C01812=1021.394,-73.795,405.018,166.174,50.269,159.076
C01813=1021.400,-73.545,405.007,166.177,50.265,159.076
C01814=1021.405,-73.295,404.997,166.180,50.261,159.076
C01815=1021.410,-73.046,404.986,166.182,50.257,159.076
C01816=1021.416,-72.796,404.976,166.185,50.253,159.075
C01817=1021.423,-72.475,404.962,166.189,50.248,159.075
C01818=1021.430,-72.155,404.949,166.193,50.243,159.075
C01819=1021.437,-71.835,404.935,166.198,50.238,159.075
C01820=1021.444,-71.515,404.921,166.201,50.233,159.074
C01821=1021.449,-71.265,404.910,166.204,50.228,159.074
C01822=1021.454,-71.015,404.900,166.207,50.225,159.074
C01823=1021.460,-70.766,404.889,166.210,50.221,159.074
C01824=1021.466,-70.516,404.878,166.213,50.217,159.073
C01825=1021.471,-70.286,404.869,166.216,50.213,159.073
C01826=1021.476,-70.056,404.859,166.219,50.209,159.073
C01827=1021.481,-69.826,404.849,166.221,50.206,159.073
C01828=1021.487,-69.597,404.839,166.224,50.202,159.073
C01829=1021.492,-69.367,404.829,166.227,50.199,159.072
C01830=1021.497,-69.138,404.820,166.229,50.195,159.072
C01831=1021.502,-68.907,404.809,166.232,50.191,159.072
C01832=1021.507,-68.677,404.800,166.235,50.187,159.072
C01833=1021.513,-68.428,404.789,166.238,50.184,159.072
C01834=1021.518,-68.178,404.778,166.241,50.180,159.071
C01835=1021.524,-67.928,404.768,166.243,50.176,159.071
C01836=1021.530,-67.679,404.757,166.247,50.171,159.071
C01837=1021.535,-67.429,404.746,166.250,50.167,159.071
C01838=1021.541,-67.180,404.735,166.253,50.164,159.071
C01839=1021.546,-66.930,404.725,166.256,50.160,159.070
C01840=1021.552,-66.680,404.714,166.259,50.155,159.070
C01841=1021.558,-66.431,404.703,166.262,50.151,159.070
C01842=1021.564,-66.181,404.692,166.265,50.147,159.070
C01843=1021.569,-65.932,404.681,166.268,50.144,159.070
C01844=1021.575,-65.681,404.670,166.272,50.139,159.069
C01845=1021.580,-65.431,404.659,166.274,50.135,159.069
C01846=1021.586,-65.182,404.648,166.277,50.131,159.069
C01847=1021.592,-64.932,404.638,166.280,50.127,159.069
C01848=1021.598,-64.683,404.627,166.282,50.123,159.068
C01849=1021.603,-64.433,404.617,166.286,50.119,159.068
C01850=1021.609,-64.183,404.606,166.289,50.115,159.068
C01851=1021.615,-63.934,404.595,166.292,50.111,159.068
C01852=1021.620,-63.684,404.584,166.294,50.107,159.067
C01853=1021.626,-63.434,404.572,166.298,50.103,159.067
C01854=1021.632,-63.184,404.561,166.301,50.099,159.067
C01855=1021.637,-62.935,404.550,166.304,50.095,159.067
C01856=1021.643,-62.685,404.539,166.306,50.090,159.066
C01857=1021.649,-62.436,404.529,166.310,50.086,159.066
C01858=1021.654,-62.186,404.518,166.313,50.083,159.066
C01859=1021.660,-61.936,404.508,166.316,50.079,159.066
C01860=1021.666,-61.686,404.496,166.318,50.075,159.066
C01861=1021.672,-61.436,404.485,166.322,50.070,159.065
C01862=1021.677,-61.187,404.474,166.325,50.066,159.065
C01863=1021.683,-60.937,404.463,166.328,50.062,159.065
C01864=1021.689,-60.688,404.452,166.330,50.058,159.064
C01865=1021.695,-60.437,404.441,166.334,50.054,159.064
C01866=1021.701,-60.188,404.430,166.337,50.050,159.064
C01867=1021.706,-59.938,404.419,166.339,50.045,159.064
C01868=1021.712,-59.689,404.408,166.343,50.041,159.064
C01869=1021.718,-59.439,404.397,166.346,50.037,159.063
C01870=1021.724,-59.189,404.386,166.349,50.033,159.063
C01871=1021.729,-58.939,404.375,166.352,50.030,159.063
C01872=1021.735,-58.690,404.364,166.355,50.025,159.063
C01873=1021.741,-58.441,404.353,166.358,50.021,159.062
C01874=1021.747,-58.190,404.342,166.361,50.017,159.062
C01875=1021.753,-57.941,404.331,166.363,50.013,159.062
C01876=1021.759,-57.691,404.320,166.367,50.009,159.062
C01877=1021.764,-57.442,404.309,166.370,50.005,159.061
C01878=1021.770,-57.191,404.297,166.373,50.000,159.061
C01879=1021.776,-56.942,404.286,166.375,49.996,159.061
C01880=1021.782,-56.693,404.275,166.379,49.992,159.061
C01881=1021.788,-56.443,404.264,166.382,49.988,159.060
C01882=1021.794,-56.193,404.253,166.384,49.984,159.060
C01883=1021.799,-55.944,404.242,166.388,49.980,159.060
C01884=1021.804,-55.694,404.230,166.391,49.975,159.060
C01885=1021.811,-55.444,404.219,166.394,49.971,159.059
C01886=1021.817,-55.194,404.208,166.396,49.967,159.059
C01887=1021.822,-54.945,404.197,166.400,49.963,159.059
C01888=1021.829,-54.695,404.185,166.403,49.959,159.059
C01889=1021.835,-54.446,404.174,166.405,49.955,159.058
C01890=1021.840,-54.196,404.164,166.409,49.950,159.058
C01891=1021.846,-53.946,404.152,166.412,49.946,159.058
C01892=1021.852,-53.696,404.141,166.414,49.942,159.057
C01893=1021.859,-53.417,404.128,166.418,49.937,159.057
C01894=1021.866,-53.138,404.116,166.421,49.932,159.057
C01895=1021.872,-52.859,404.103,166.424,49.928,159.057
C01896=1021.879,-52.579,404.091,166.427,49.923,159.056
C01897=1021.885,-52.330,404.079,166.431,49.919,159.056
C01898=1021.890,-52.080,404.068,166.434,49.915,159.056
C01899=1021.897,-51.830,404.057,166.437,49.911,159.055
C01900=1021.902,-51.580,404.045,166.439,49.907,159.055
C01901=1021.908,-51.331,404.033,166.443,49.902,159.055
C01902=1021.914,-51.081,404.023,166.446,49.898,159.055
C01903=1021.920,-50.832,404.012,166.448,49.894,159.054
C01904=1021.926,-50.582,403.999,166.451,49.890,159.054
C01905=1021.932,-50.332,403.988,166.455,49.886,159.054
C01906=1021.937,-50.082,403.976,166.458,49.882,159.054
C01907=1021.943,-49.833,403.965,166.460,49.878,159.053
C01908=1021.949,-49.583,403.953,166.463,49.874,159.053
C01909=1021.955,-49.334,403.941,166.466,49.870,159.053
C01910=1021.960,-49.084,403.930,166.469,49.866,159.053
C01911=1021.966,-48.834,403.917,166.473,49.862,159.052
C01912=1021.971,-48.584,403.906,166.475,49.858,159.052
C01913=1021.977,-48.335,403.894,166.478,49.854,159.052
C01914=1021.983,-48.085,403.883,166.481,49.850,159.052
C01915=1021.989,-47.835,403.870,166.484,49.846,159.051
C01916=1021.995,-47.586,403.860,166.486,49.842,159.051
C01917=1022.000,-47.337,403.847,166.490,49.838,159.051
C01918=1022.006,-47.086,403.836,166.493,49.834,159.051
C01919=1022.012,-46.837,403.824,166.496,49.830,159.050
C01920=1022.017,-46.587,403.812,166.498,49.826,159.050
C01921=1022.023,-46.338,403.801,166.501,49.822,159.050
C01922=1022.029,-46.088,403.788,166.504,49.818,159.050
C01923=1022.035,-45.838,403.777,166.508,49.814,159.050
C01924=1022.041,-45.589,403.765,166.511,49.810,159.049
C01925=1022.047,-45.339,403.754,166.513,49.806,159.049
C01926=1022.053,-45.089,403.741,166.516,49.802,159.049
C01927=1022.059,-44.840,403.730,166.519,49.798,159.048
C01928=1022.064,-44.590,403.718,166.521,49.794,159.048
C01929=1022.070,-44.341,403.705,166.525,49.789,159.048
C01930=1022.076,-44.090,403.694,166.528,49.785,159.048
C01931=1022.081,-43.841,403.682,166.531,49.781,159.047
C01932=1022.088,-43.592,403.670,166.533,49.777,159.047
C01933=1022.093,-43.341,403.658,166.536,49.773,159.047
C01934=1022.099,-43.092,403.647,166.540,49.770,159.047
C01935=1022.105,-42.842,403.634,166.543,49.766,159.046
C01936=1022.110,-42.593,403.623,166.546,49.762,159.046
C01937=1022.117,-42.343,403.611,166.548,49.758,159.046
C01938=1022.122,-42.094,403.599,166.551,49.753,159.045
C01939=1022.129,-41.844,403.587,166.554,49.749,159.045
C01940=1022.134,-41.594,403.575,166.558,49.745,159.045
C01941=1022.140,-41.345,403.563,166.560,49.741,159.045
C01942=1022.147,-41.095,403.551,166.563,49.737,159.044
C01943=1022.152,-40.845,403.539,166.566,49.733,159.044
C01944=1022.158,-40.596,403.527,166.568,49.729,159.044
C01945=1022.163,-40.346,403.515,166.572,49.725,159.044
C01946=1022.170,-40.097,403.503,166.575,49.721,159.043
C01947=1022.176,-39.846,403.491,166.578,49.717,159.043
C01948=1022.181,-39.597,403.479,166.580,49.713,159.043
C01949=1022.188,-39.348,403.467,166.583,49.708,159.042
C01950=1022.194,-39.098,403.454,166.587,49.704,159.042
C01951=1022.199,-38.849,403.442,166.589,49.700,159.042
C01952=1022.204,-38.598,403.430,166.592,49.696,159.042
C01953=1022.210,-38.348,403.418,166.595,49.692,159.041
C01954=1022.216,-38.099,403.406,166.598,49.688,159.041
C01955=1022.222,-37.849,403.394,166.601,49.685,159.041
C01956=1022.228,-37.600,403.381,166.603,49.681,159.041
C01957=1022.234,-37.321,403.367,166.607,49.676,159.040
C01958=1022.241,-37.043,403.354,166.610,49.672,159.040
C01959=1022.248,-36.763,403.341,166.613,49.667,159.040
C01960=1022.253,-36.484,403.327,166.617,49.662,159.039
C01961=1022.259,-36.234,403.314,166.620,49.659,159.039
C01962=1022.265,-35.984,403.301,166.623,49.655,159.039
C01963=1022.271,-35.735,403.289,166.625,49.651,159.039
C01964=1022.277,-35.486,403.277,166.628,49.647,159.038
C01965=1022.283,-35.236,403.265,166.631,49.643,159.038
C01966=1022.288,-34.987,403.253,166.633,49.639,159.038
C01967=1022.294,-34.737,403.240,166.636,49.635,159.037
C01968=1022.300,-34.487,403.227,166.640,49.630,159.037
C01969=1022.306,-34.237,403.215,166.643,49.626,159.037
C01970=1022.312,-33.988,403.203,166.645,49.622,159.037
C01971=1022.318,-33.738,403.191,166.648,49.618,159.036
C01972=1022.324,-33.488,403.178,166.651,49.615,159.036
C01973=1022.330,-33.238,403.166,166.654,49.611,159.036
C01974=1022.336,-32.990,403.153,166.657,49.607,159.036
C01975=1022.341,-32.740,403.140,166.659,49.603,159.035
C01976=1022.347,-32.490,403.128,166.663,49.599,159.035
C01977=1022.353,-32.240,403.115,166.666,49.595,159.035
C01978=1022.359,-31.991,403.103,166.669,49.591,159.035
C01979=1022.365,-31.742,403.091,166.671,49.587,159.034
C01980=1022.371,-31.492,403.078,166.674,49.583,159.034
C01981=1022.377,-31.242,403.066,166.677,49.579,159.034
C01982=1022.382,-30.993,403.054,166.679,49.575,159.033
C01983=1022.388,-30.743,403.041,166.682,49.570,159.033
C01984=1022.395,-30.493,403.028,166.686,49.566,159.033
C01985=1022.400,-30.244,403.015,166.689,49.562,159.033
C01986=1022.406,-29.994,403.003,166.691,49.558,159.032
C01987=1022.412,-29.745,402.991,166.694,49.554,159.032
C01988=1022.418,-29.495,402.979,166.697,49.550,159.032
C01989=1022.424,-29.245,402.966,166.700,49.546,159.031
C01990=1022.430,-28.996,402.953,166.702,49.542,159.031
C01991=1022.436,-28.746,402.940,166.706,49.538,159.031
C01992=1022.442,-28.496,402.928,166.709,49.534,159.031
C01993=1022.448,-28.247,402.915,166.711,49.530,159.030
C01994=1022.453,-27.997,402.903,166.714,49.526,159.030
C01995=1022.460,-27.748,402.890,166.717,49.522,159.030
C01996=1022.466,-27.498,402.878,166.720,49.518,159.029
C01997=1022.471,-27.248,402.864,166.722,49.514,159.029
C01998=1022.477,-26.998,402.852,166.725,49.510,159.029
C01999=1022.484,-26.749,402.839,166.728,49.506,159.028
C02000=1022.489,-26.499,402.826,166.731,49.502,159.028
C02001=1022.495,-26.250,402.814,166.734,49.497,159.028
C02002=1022.501,-26.000,402.801,166.737,49.493,159.028
C02003=1022.506,-25.750,402.787,166.740,49.490,159.028
C02004=1022.512,-25.501,402.774,166.743,49.486,159.027
C02005=1022.518,-25.251,402.762,166.746,49.482,159.027
C02006=1022.524,-25.001,402.749,166.748,49.478,159.027
C02007=1022.530,-24.752,402.736,166.751,49.474,159.026
C02008=1022.536,-24.502,402.723,166.754,49.470,159.026
C02009=1022.541,-24.253,402.710,166.757,49.466,159.026
C02010=1022.547,-24.003,402.697,166.759,49.462,159.025
C02011=1022.553,-23.754,402.684,166.762,49.458,159.025
C02012=1022.559,-23.504,402.671,166.765,49.454,159.025
C02013=1022.565,-23.255,402.658,166.768,49.450,159.024
C02014=1022.571,-23.005,402.646,166.770,49.446,159.024
C02015=1022.577,-22.755,402.632,166.773,49.443,159.024
C02016=1022.583,-22.506,402.619,166.776,49.439,159.024
C02017=1022.589,-22.256,402.607,166.779,49.435,159.023
C02018=1022.595,-22.006,402.593,166.783,49.430,159.023
C02019=1022.601,-21.756,402.581,166.785,49.426,159.023
C02020=1022.606,-21.507,402.567,166.788,49.422,159.023
C02021=1022.613,-21.228,402.553,166.790,49.418,159.022
C02022=1022.620,-20.947,402.538,166.794,49.413,159.022
C02023=1022.626,-20.668,402.523,166.797,49.409,159.021
C02024=1022.633,-20.388,402.509,166.800,49.404,159.021
C02025=1022.639,-20.138,402.496,166.803,49.400,159.021
C02026=1022.645,-19.889,402.483,166.806,49.396,159.021
C02027=1022.651,-19.639,402.470,166.809,49.392,159.020
C02028=1022.657,-19.389,402.456,166.811,49.388,159.020
C02029=1022.663,-19.140,402.444,166.814,49.384,159.020
C02030=1022.669,-18.890,402.430,166.817,49.380,159.019
C02031=1022.675,-18.641,402.417,166.820,49.376,159.019
C02032=1022.680,-18.391,402.404,166.823,49.372,159.019
C02033=1022.687,-18.142,402.391,166.826,49.368,159.019
C02034=1022.693,-17.892,402.378,166.829,49.364,159.018
C02035=1022.699,-17.642,402.365,166.832,49.360,159.018
C02036=1022.705,-17.393,402.352,166.834,49.356,159.018
C02037=1022.711,-17.143,402.339,166.837,49.352,159.017
C02038=1022.716,-16.894,402.325,166.840,49.348,159.017
C02039=1022.722,-16.644,402.312,166.842,49.343,159.017
C02040=1022.728,-16.395,402.299,166.845,49.339,159.016
C02041=1022.735,-16.145,402.286,166.848,49.335,159.016
C02042=1022.741,-15.896,402.273,166.850,49.331,159.016
C02043=1022.746,-15.646,402.260,166.853,49.327,159.015
C02044=1022.752,-15.397,402.247,166.856,49.323,159.015
C02045=1022.758,-15.147,402.233,166.859,49.319,159.015
C02046=1022.764,-14.898,402.219,166.862,49.316,159.015
C02047=1022.769,-14.648,402.206,166.864,49.312,159.014
C02048=1022.776,-14.398,402.193,166.867,49.308,159.014
C02049=1022.781,-14.148,402.179,166.870,49.304,159.014
C02050=1022.788,-13.899,402.165,166.873,49.300,159.013
C02051=1022.793,-13.649,402.152,166.875,49.296,159.013
C02052=1022.799,-13.400,402.138,166.878,49.292,159.013
C02053=1022.805,-13.151,402.125,166.881,49.288,159.012
C02054=1022.811,-12.900,402.112,166.884,49.284,159.012
C02055=1022.817,-12.651,402.099,166.886,49.280,159.012
C02056=1022.822,-12.402,402.085,166.889,49.276,159.011
C02057=1022.829,-12.152,402.072,166.892,49.272,159.011
C02058=1022.835,-11.902,402.057,166.895,49.268,159.011
C02059=1022.841,-11.653,402.044,166.897,49.264,159.010
C02060=1022.846,-11.403,402.030,166.900,49.260,159.010
C02061=1022.853,-11.154,402.017,166.903,49.256,159.010
C02062=1022.858,-10.904,402.003,166.906,49.252,159.010
C02063=1022.864,-10.655,401.990,166.908,49.248,159.009
C02064=1022.869,-10.405,401.977,166.911,49.244,159.009
C02065=1022.876,-10.155,401.963,166.915,49.240,159.009
C02066=1022.882,-9.905,401.949,166.918,49.236,159.008
C02067=1022.888,-9.656,401.936,166.920,49.232,159.008
C02068=1022.893,-9.406,401.922,166.923,49.228,159.008
C02069=1022.900,-9.157,401.909,166.926,49.224,159.007
C02070=1022.905,-8.908,401.895,166.929,49.220,159.007
C02071=1022.912,-8.658,401.881,166.931,49.216,159.007
C02072=1022.918,-8.408,401.868,166.934,49.212,159.007
C02073=1022.924,-8.159,401.854,166.937,49.208,159.006
C02074=1022.930,-7.910,401.841,166.940,49.204,159.006
C02075=1022.935,-7.660,401.827,166.942,49.200,159.006
C02076=1022.942,-7.410,401.813,166.945,49.196,159.005
C02077=1022.948,-7.160,401.799,166.948,49.192,159.005
C02078=1022.954,-6.911,401.786,166.951,49.188,159.005
C02079=1022.959,-6.662,401.772,166.953,49.184,159.004
C02080=1022.966,-6.412,401.759,166.956,49.180,159.004
C02081=1022.972,-6.162,401.745,166.959,49.176,159.004
C02082=1022.978,-5.913,401.732,166.962,49.172,159.003
C02083=1022.983,-5.663,401.718,166.964,49.169,159.003
C02084=1022.990,-5.414,401.703,166.967,49.165,159.003
C02085=1022.997,-5.132,401.688,166.970,49.160,159.002
C02086=1023.003,-4.851,401.672,166.973,49.155,159.002
C02087=1023.010,-4.569,401.657,166.977,49.151,159.002
C02088=1023.017,-4.288,401.641,166.979,49.146,159.001
C02089=1023.023,-4.039,401.628,166.982,49.142,159.001
C02090=1023.029,-3.788,401.614,166.985,49.138,159.001
C02091=1023.034,-3.539,401.600,166.987,49.134,159.000
C02092=1023.040,-3.289,401.586,166.990,49.130,159.000
C02093=1023.046,-3.040,401.571,166.993,49.127,159.000
C02094=1023.052,-2.790,401.557,166.996,49.123,158.999
C02095=1023.058,-2.541,401.544,166.999,49.119,158.999
C02096=1023.064,-2.292,401.529,167.002,49.115,158.999
C02097=1023.070,-2.041,401.515,167.003,49.111,158.998
C02098=1023.075,-1.792,401.501,167.006,49.107,158.998
C02099=1023.081,-1.543,401.487,167.009,49.103,158.998
C02100=1023.087,-1.293,401.472,167.012,49.099,158.997
C02101=1023.093,-1.043,401.459,167.014,49.095,158.997
C02102=1023.099,-0.794,401.445,167.017,49.091,158.997
C02103=1023.105,-0.545,401.431,167.020,49.087,158.997
C02104=1023.111,-0.295,401.416,167.023,49.083,158.996
C02105=1023.117,-0.046,401.402,167.026,49.080,158.996
C02106=1023.122,0.204,401.388,167.028,49.076,158.996
C02107=1023.128,0.454,401.374,167.031,49.072,158.995
C02108=1023.134,0.703,401.359,167.034,49.068,158.995
C02109=1023.140,0.952,401.346,167.037,49.064,158.995
C02110=1023.146,1.203,401.332,167.039,49.060,158.994
C02111=1023.152,1.452,401.317,167.041,49.057,158.994
C02112=1023.157,1.701,401.303,167.044,49.053,158.994
C02113=1023.164,1.951,401.288,167.047,49.049,158.993
C02114=1023.169,2.200,401.274,167.049,49.045,158.993
C02115=1023.176,2.450,401.259,167.052,49.041,158.993
C02116=1023.182,2.699,401.246,167.055,49.037,158.992
C02117=1023.187,2.949,401.232,167.058,49.033,158.992
C02118=1023.194,3.199,401.217,167.060,49.029,158.992
C02119=1023.199,3.448,401.204,167.063,49.025,158.991
C02120=1023.205,3.697,401.189,167.066,49.021,158.991
C02121=1023.211,3.947,401.175,167.069,49.017,158.991
C02122=1023.217,4.196,401.160,167.072,49.013,158.991
C02123=1023.223,4.447,401.146,167.074,49.009,158.990
C02124=1023.229,4.695,401.132,167.077,49.005,158.990
C02125=1023.236,4.946,401.118,167.080,49.001,158.990
C02126=1023.241,5.195,401.103,167.083,48.997,158.989
C02127=1023.247,5.444,401.089,167.084,48.994,158.989
C02128=1023.253,5.694,401.074,167.087,48.990,158.989
C02129=1023.259,5.943,401.060,167.089,48.985,158.988
C02130=1023.265,6.193,401.046,167.092,48.981,158.988
C02131=1023.271,6.443,401.032,167.095,48.977,158.987
C02132=1023.278,6.692,401.017,167.098,48.973,158.987
C02133=1023.283,6.941,401.003,167.101,48.969,158.987
C02134=1023.289,7.190,400.989,167.103,48.965,158.986
C02135=1023.295,7.440,400.974,167.106,48.961,158.986
C02136=1023.301,7.690,400.960,167.109,48.957,158.986
C02137=1023.307,7.939,400.945,167.112,48.953,158.985
C02138=1023.313,8.189,400.931,167.114,48.950,158.985
C02139=1023.319,8.439,400.916,167.117,48.946,158.985
C02140=1023.325,8.688,400.902,167.120,48.941,158.984
C02141=1023.332,8.937,400.888,167.122,48.937,158.984
C02142=1023.337,9.186,400.873,167.125,48.933,158.984
C02143=1023.343,9.437,400.859,167.128,48.929,158.983
C02144=1023.349,9.686,400.845,167.131,48.925,158.983
C02145=1023.356,9.935,400.830,167.133,48.921,158.983
C02146=1023.361,10.185,400.816,167.136,48.917,158.982
C02147=1023.367,10.435,400.801,167.139,48.913,158.982
C02148=1023.373,10.684,400.786,167.141,48.909,158.982
C02149=1023.380,10.967,400.770,167.144,48.905,158.981
C02150=1023.387,11.250,400.754,167.148,48.900,158.981
C02151=1023.394,11.534,400.737,167.150,48.895,158.980
C02152=1023.402,11.817,400.721,167.153,48.890,158.980
C02153=1023.407,12.066,400.706,167.156,48.886,158.980
C02154=1023.413,12.317,400.692,167.159,48.882,158.979
C02155=1023.420,12.566,400.677,167.162,48.878,158.979
C02156=1023.426,12.815,400.663,167.164,48.875,158.979
C02157=1023.432,13.066,400.648,167.166,48.871,158.978
C02158=1023.437,13.314,400.634,167.169,48.866,158.978
C02159=1023.444,13.564,400.619,167.172,48.862,158.977
C02160=1023.450,13.814,400.604,167.174,48.858,158.977
C02161=1023.456,14.063,400.589,167.177,48.854,158.977
C02162=1023.462,14.313,400.575,167.180,48.850,158.976
C02163=1023.467,14.562,400.560,167.183,48.846,158.976
C02164=1023.473,14.812,400.545,167.185,48.843,158.976
C02165=1023.479,15.061,400.530,167.188,48.839,158.975
C02166=1023.486,15.311,400.515,167.191,48.835,158.975
C02167=1023.492,15.560,400.500,167.194,48.831,158.975
C02168=1023.498,15.809,400.486,167.195,48.827,158.974
C02169=1023.503,16.059,400.470,167.198,48.823,158.974
C02170=1023.509,16.308,400.456,167.201,48.819,158.974
C02171=1023.515,16.558,400.442,167.204,48.815,158.973
C02172=1023.522,16.808,400.427,167.207,48.811,158.973
C02173=1023.527,17.057,400.412,167.209,48.807,158.973
C02174=1023.533,17.307,400.396,167.212,48.803,158.972
C02175=1023.539,17.556,400.382,167.215,48.799,158.972
C02176=1023.545,17.806,400.367,167.217,48.795,158.972
C02177=1023.552,18.055,400.352,167.220,48.791,158.971
C02178=1023.557,18.304,400.337,167.222,48.787,158.971
C02179=1023.563,18.554,400.322,167.225,48.783,158.971
C02180=1023.569,18.804,400.307,167.227,48.779,158.970
C02181=1023.575,19.053,400.292,167.230,48.776,158.970
C02182=1023.582,19.302,400.277,167.233,48.772,158.970
C02183=1023.588,19.552,400.262,167.236,48.768,158.969
C02184=1023.593,19.801,400.247,167.238,48.763,158.969
C02185=1023.599,20.051,400.232,167.241,48.759,158.968
C02186=1023.606,20.301,400.217,167.243,48.755,158.968
C02187=1023.611,20.550,400.202,167.245,48.752,158.968
C02188=1023.617,20.800,400.187,167.248,48.748,158.967
C02189=1023.624,21.049,400.172,167.251,48.744,158.967
C02190=1023.629,21.298,400.156,167.254,48.740,158.967
C02191=1023.635,21.548,400.142,167.257,48.736,158.966
C02192=1023.642,21.797,400.127,167.259,48.732,158.966
C02193=1023.647,22.046,400.111,167.262,48.728,158.966
C02194=1023.653,22.296,400.096,167.264,48.724,158.965
C02195=1023.659,22.546,400.081,167.267,48.720,158.965
C02196=1023.665,22.795,400.066,167.269,48.716,158.965
C02197=1023.671,23.044,400.051,167.272,48.713,158.964
C02198=1023.677,23.294,400.035,167.275,48.708,158.964
C02199=1023.683,23.544,400.020,167.277,48.704,158.963
C02200=1023.689,23.793,400.006,167.280,48.700,158.963
C02201=1023.695,24.043,399.990,167.283,48.696,158.963
C02202=1023.701,24.292,399.975,167.285,48.693,158.962
C02203=1023.707,24.541,399.960,167.288,48.689,158.962
C02204=1023.713,24.791,399.944,167.290,48.685,158.962
C02205=1023.719,25.040,399.929,167.293,48.681,158.961
C02206=1023.726,25.290,399.914,167.296,48.676,158.961
C02207=1023.731,25.539,399.899,167.298,48.672,158.961
C02208=1023.737,25.788,399.884,167.301,48.668,158.960
C02209=1023.743,26.038,399.868,167.304,48.664,158.960
C02210=1023.749,26.288,399.853,167.307,48.661,158.960
C02211=1023.755,26.537,399.838,167.308,48.657,158.959
C02212=1023.761,26.786,399.822,167.311,48.653,158.959
C02213=1023.768,27.071,399.805,167.315,48.648,158.958
C02214=1023.775,27.356,399.788,167.317,48.643,158.958
C02215=1023.782,27.641,399.770,167.321,48.639,158.958
C02216=1023.788,27.926,399.753,167.323,48.635,158.957
C02217=1023.795,28.175,399.737,167.326,48.631,158.957
C02218=1023.801,28.425,399.722,167.329,48.627,158.956
C02219=1023.806,28.675,399.706,167.331,48.623,158.956
C02220=1023.813,28.923,399.691,167.334,48.619,158.956
C02221=1023.818,29.173,399.675,167.336,48.615,158.955
C02222=1023.825,29.422,399.659,167.339,48.611,158.955
C02223=1023.831,29.672,399.644,167.342,48.608,158.955
C02224=1023.836,29.922,399.628,167.344,48.603,158.954
C02225=1023.842,30.170,399.613,167.346,48.599,158.954
C02226=1023.848,30.420,399.598,167.349,48.595,158.953
C02227=1023.855,30.669,399.582,167.352,48.591,158.953
C02228=1023.860,30.919,399.566,167.355,48.588,158.953
C02229=1023.866,31.169,399.550,167.357,48.584,158.952
C02230=1023.873,31.418,399.535,167.360,48.580,158.952
C02231=1023.878,31.667,399.519,167.362,48.576,158.952
C02232=1023.884,31.917,399.504,167.365,48.572,158.951
C02233=1023.890,32.166,399.488,167.367,48.568,158.951
C02234=1023.896,32.416,399.473,167.370,48.564,158.951
C02235=1023.903,32.665,399.457,167.373,48.560,158.950
C02236=1023.908,32.915,399.441,167.375,48.556,158.950
C02237=1023.914,33.163,399.426,167.378,48.552,158.950
C02238=1023.920,33.413,399.410,167.380,48.548,158.949
C02239=1023.926,33.663,399.394,167.383,48.544,158.949
C02240=1023.932,33.912,399.379,167.386,48.541,158.948
C02241=1023.938,34.162,399.363,167.388,48.537,158.948
C02242=1023.944,34.412,399.347,167.391,48.532,158.948
C02243=1023.951,34.661,399.332,167.394,48.528,158.947
C02244=1023.956,34.911,399.316,167.395,48.525,158.947
C02245=1023.963,35.160,399.301,167.398,48.521,158.946
C02246=1023.968,35.409,399.285,167.401,48.517,158.946
C02247=1023.974,35.658,399.269,167.404,48.513,158.946
C02248=1023.981,35.907,399.254,167.406,48.508,158.945
C02249=1023.986,36.157,399.238,167.409,48.504,158.945
C02250=1023.993,36.406,399.222,167.412,48.500,158.945
C02251=1023.999,36.656,399.207,167.415,48.497,158.944
C02252=1024.005,36.906,399.191,167.416,48.493,158.944
C02253=1024.010,37.155,399.174,167.419,48.489,158.944
C02254=1024.017,37.405,399.159,167.422,48.485,158.943
C02255=1024.023,37.654,399.143,167.425,48.481,158.943
C02256=1024.029,37.903,399.127,167.428,48.477,158.943
C02257=1024.034,38.153,399.111,167.429,48.473,158.942
C02258=1024.040,38.402,399.095,167.432,48.469,158.942
C02259=1024.046,38.651,399.079,167.435,48.465,158.941
C02260=1024.052,38.901,399.063,167.437,48.461,158.941
C02261=1024.058,39.150,399.048,167.440,48.457,158.941
C02262=1024.064,39.400,399.032,167.442,48.454,158.940
C02263=1024.070,39.649,399.015,167.445,48.450,158.940
C02264=1024.076,39.898,398.999,167.448,48.446,158.940
C02265=1024.082,40.148,398.983,167.450,48.442,158.939
C02266=1024.087,40.398,398.967,167.453,48.438,158.939
C02267=1024.093,40.647,398.951,167.455,48.435,158.938
C02268=1024.100,40.896,398.935,167.457,48.430,158.938
C02269=1024.106,41.145,398.919,167.460,48.426,158.938
C02270=1024.112,41.395,398.904,167.463,48.422,158.937
C02271=1024.118,41.645,398.887,167.466,48.418,158.937
C02272=1024.124,41.894,398.871,167.469,48.415,158.937
C02273=1024.130,42.143,398.855,167.470,48.411,158.936
C02274=1024.136,42.393,398.839,167.473,48.407,158.936
C02275=1024.141,42.642,398.822,167.476,48.403,158.935
C02276=1024.147,42.891,398.806,167.479,48.399,158.935
C02277=1024.154,43.176,398.788,167.481,48.395,158.935
C02278=1024.161,43.461,398.769,167.484,48.391,158.934
C02279=1024.168,43.747,398.751,167.488,48.386,158.934
C02280=1024.174,44.031,398.732,167.490,48.381,158.933
C02281=1024.180,44.280,398.716,167.493,48.377,158.933
C02282=1024.186,44.530,398.700,167.495,48.374,158.933
C02283=1024.192,44.779,398.684,167.498,48.370,158.932
C02284=1024.197,45.029,398.667,167.500,48.366,158.932
C02285=1024.203,45.278,398.650,167.503,48.362,158.932
C02286=1024.209,45.527,398.634,167.505,48.359,158.931
C02287=1024.215,45.777,398.618,167.508,48.355,158.931
C02288=1024.221,46.026,398.602,167.511,48.351,158.930
C02289=1024.227,46.275,398.585,167.513,48.347,158.930
C02290=1024.233,46.525,398.569,167.515,48.343,158.930
C02291=1024.238,46.774,398.552,167.518,48.339,158.929
C02292=1024.244,47.024,398.536,167.521,48.336,158.929
C02293=1024.250,47.272,398.519,167.524,48.332,158.929
C02294=1024.256,47.522,398.503,167.525,48.328,158.928
C02295=1024.262,47.771,398.487,167.528,48.324,158.928
C02296=1024.269,48.021,398.470,167.531,48.320,158.928
C02297=1024.274,48.271,398.453,167.534,48.317,158.927
C02298=1024.280,48.520,398.437,167.535,48.313,158.927
C02299=1024.286,48.770,398.421,167.538,48.309,158.926
C02300=1024.292,49.019,398.404,167.541,48.305,158.926
C02301=1024.298,49.268,398.388,167.544,48.301,158.926
C02302=1024.304,49.518,398.372,167.547,48.297,158.925
C02303=1024.310,49.766,398.355,167.549,48.294,158.925
C02304=1024.315,50.016,398.338,167.551,48.289,158.924
C02305=1024.321,50.265,398.322,167.554,48.285,158.924
C02306=1024.327,50.515,398.305,167.557,48.281,158.924
C02307=1024.333,50.764,398.289,167.558,48.278,158.923
C02308=1024.340,51.014,398.273,167.561,48.274,158.923
C02309=1024.345,51.263,398.256,167.564,48.270,158.923
C02310=1024.351,51.512,398.239,167.567,48.266,158.922
C02311=1024.357,51.762,398.222,167.570,48.262,158.922
C02312=1024.363,52.011,398.206,167.571,48.259,158.922
C02313=1024.369,52.261,398.190,167.574,48.254,158.921
C02314=1024.375,52.510,398.174,167.577,48.250,158.921
C02315=1024.382,52.759,398.156,167.580,48.247,158.920
C02316=1024.387,53.009,398.140,167.582,48.243,158.920
C02317=1024.393,53.258,398.123,167.584,48.239,158.920
C02318=1024.399,53.508,398.107,167.587,48.235,158.919
C02319=1024.405,53.757,398.091,167.589,48.231,158.919
C02320=1024.411,54.006,398.074,167.592,48.227,158.918
C02321=1024.417,54.256,398.057,167.595,48.223,158.918
C02322=1024.423,54.505,398.040,167.597,48.219,158.918
C02323=1024.429,54.755,398.024,167.600,48.215,158.917
C02324=1024.435,55.004,398.007,167.602,48.212,158.917
C02325=1024.441,55.253,397.991,167.605,48.207,158.916
C02326=1024.447,55.502,397.975,167.608,48.203,158.916
C02327=1024.453,55.752,397.957,167.610,48.200,158.916
C02328=1024.459,56.001,397.940,167.612,48.196,158.915
C02329=1024.465,56.251,397.924,167.615,48.192,158.915
C02330=1024.471,56.500,397.908,167.618,48.187,158.914
C02331=1024.477,56.749,397.891,167.621,48.183,158.914
C02332=1024.483,56.999,397.874,167.623,48.180,158.914
C02333=1024.489,57.248,397.857,167.625,48.176,158.913
C02334=1024.495,57.497,397.840,167.628,48.172,158.913
C02335=1024.501,57.747,397.824,167.630,48.168,158.912
C02336=1024.508,57.997,397.808,167.633,48.164,158.912
C02337=1024.514,58.245,397.791,167.636,48.160,158.912
C02338=1024.519,58.495,397.774,167.638,48.156,158.911
C02339=1024.525,58.744,397.758,167.640,48.152,158.911
C02340=1024.532,58.994,397.740,167.643,48.148,158.911
C02341=1024.538,59.278,397.722,167.647,48.143,158.910
C02342=1024.545,59.563,397.703,167.649,48.138,158.910
C02343=1024.553,59.847,397.683,167.652,48.134,158.909
C02344=1024.559,60.131,397.664,167.656,48.130,158.909
C02345=1024.565,60.382,397.647,167.658,48.125,158.908
C02346=1024.571,60.630,397.630,167.660,48.122,158.908
C02347=1024.577,60.880,397.614,167.663,48.118,158.907
C02348=1024.584,61.130,397.597,167.665,48.113,158.907
C02349=1024.590,61.379,397.580,167.668,48.109,158.907
C02350=1024.595,61.628,397.563,167.671,48.106,158.906
C02351=1024.602,61.877,397.546,167.674,48.102,158.906
C02352=1024.608,62.127,397.530,167.675,48.097,158.905
C02353=1024.615,62.376,397.513,167.678,48.094,158.905
C02354=1024.620,62.625,397.497,167.681,48.090,158.905
C02355=1024.627,62.875,397.479,167.683,48.085,158.904
C02356=1024.633,63.124,397.462,167.686,48.081,158.904
C02357=1024.639,63.373,397.445,167.689,48.078,158.903
C02358=1024.645,63.623,397.428,167.691,48.074,158.903
C02359=1024.651,63.872,397.411,167.694,48.070,158.903
C02360=1024.657,64.122,397.394,167.696,48.066,158.902
C02361=1024.663,64.371,397.377,167.699,48.062,158.902
C02362=1024.668,64.621,397.360,167.702,48.058,158.901
C02363=1024.674,64.869,397.343,167.703,48.054,158.901
C02364=1024.681,65.119,397.325,167.706,48.050,158.901
C02365=1024.686,65.369,397.309,167.709,48.047,158.900
C02366=1024.692,65.618,397.291,167.712,48.042,158.900
C02367=1024.699,65.867,397.274,167.714,48.038,158.899
C02368=1024.704,66.117,397.257,167.716,48.035,158.899
C02369=1024.711,66.366,397.240,167.719,48.031,158.899
C02370=1024.716,66.615,397.222,167.722,48.027,158.898
C02371=1024.722,66.864,397.206,167.725,48.023,158.898
C02372=1024.729,67.114,397.188,167.726,48.019,158.897
C02373=1024.734,67.363,397.171,167.729,48.015,158.897
C02374=1024.740,67.612,397.154,167.732,48.011,158.897
C02375=1024.746,67.862,397.136,167.735,48.007,158.896
C02376=1024.752,68.111,397.119,167.738,48.003,158.896
C02377=1024.758,68.360,397.102,167.739,48.000,158.896
C02378=1024.764,68.610,397.085,167.742,47.995,158.895
C02379=1024.770,68.859,397.068,167.745,47.992,158.895
C02380=1024.776,69.109,397.050,167.748,47.988,158.894
C02381=1024.782,69.358,397.033,167.749,47.984,158.894
C02382=1024.788,69.607,397.015,167.752,47.980,158.894
C02383=1024.794,69.857,396.998,167.755,47.976,158.893
C02384=1024.799,70.106,396.980,167.758,47.973,158.893
C02385=1024.805,70.355,396.963,167.761,47.969,158.893
C02386=1024.812,70.605,396.945,167.762,47.965,158.892
C02387=1024.817,70.854,396.928,167.765,47.961,158.892
C02388=1024.824,71.103,396.911,167.768,47.957,158.891
C02389=1024.829,71.352,396.893,167.771,47.953,158.891
C02390=1024.835,71.602,396.876,167.772,47.949,158.890
C02391=1024.841,71.851,396.858,167.775,47.946,158.890
C02392=1024.847,72.100,396.841,167.778,47.942,158.890
C02393=1024.853,72.350,396.823,167.781,47.938,158.889
C02394=1024.859,72.599,396.806,167.782,47.934,158.889
C02395=1024.866,72.848,396.788,167.785,47.930,158.888
C02396=1024.871,73.097,396.771,167.788,47.926,158.888
C02397=1024.877,73.347,396.753,167.791,47.922,158.888
C02398=1024.883,73.596,396.735,167.794,47.918,158.887
C02399=1024.889,73.845,396.718,167.796,47.915,158.887
C02400=1024.895,74.095,396.700,167.798,47.910,158.886
C02401=1024.901,74.344,396.683,167.801,47.906,158.886
C02402=1024.906,74.594,396.666,167.804,47.903,158.886
C02403=1024.913,74.843,396.649,167.806,47.899,158.885
C02404=1024.919,75.093,396.631,167.808,47.895,158.885
C02405=1024.925,75.377,396.610,167.812,47.890,158.884
C02406=1024.932,75.661,396.590,167.814,47.886,158.884
C02407=1024.939,75.945,396.571,167.817,47.881,158.883
C02408=1024.946,76.229,396.550,167.821,47.877,158.883
C02409=1024.952,76.479,396.532,167.822,47.873,158.883
C02410=1024.958,76.728,396.514,167.825,47.869,158.882
C02411=1024.964,76.978,396.497,167.828,47.865,158.882
C02412=1024.970,77.227,396.479,167.831,47.862,158.882
C02413=1024.976,77.476,396.461,167.833,47.858,158.881
C02414=1024.982,77.725,396.444,167.836,47.854,158.881
C02415=1024.988,77.975,396.426,167.838,47.850,158.880
C02416=1024.993,78.224,396.408,167.841,47.847,158.880
C02417=1024.999,78.474,396.390,167.843,47.843,158.880
C02418=1025.005,78.723,396.373,167.846,47.839,158.879
C02419=1025.011,78.972,396.354,167.848,47.835,158.879
C02420=1025.017,79.221,396.337,167.851,47.831,158.878
C02421=1025.023,79.471,396.319,167.853,47.827,158.878
C02422=1025.028,79.720,396.301,167.856,47.823,158.878
C02423=1025.035,79.970,396.283,167.859,47.820,158.877
C02424=1025.040,80.218,396.265,167.862,47.816,158.877
C02425=1025.047,80.468,396.247,167.863,47.812,158.876
C02426=1025.052,80.717,396.229,167.866,47.808,158.876
C02427=1025.058,80.967,396.212,167.869,47.805,158.876
C02428=1025.064,81.216,396.194,167.872,47.801,158.875
C02429=1025.070,81.465,396.175,167.873,47.797,158.875
C02430=1025.076,81.714,396.158,167.876,47.793,158.874
C02431=1025.081,81.964,396.139,167.879,47.789,158.874
C02432=1025.087,82.213,396.122,167.882,47.785,158.874
C02433=1025.093,82.462,396.103,167.885,47.781,158.873
C02434=1025.099,82.712,396.085,167.887,47.778,158.873
C02435=1025.105,82.961,396.067,167.889,47.774,158.873
C02436=1025.111,83.210,396.050,167.892,47.770,158.872
C02437=1025.117,83.459,396.031,167.895,47.766,158.872
C02438=1025.123,83.709,396.013,167.897,47.762,158.871
C02439=1025.128,83.958,395.996,167.899,47.758,158.871
C02440=1025.135,84.207,395.977,167.902,47.755,158.871
C02441=1025.141,84.457,395.959,167.905,47.751,158.870
C02442=1025.146,84.706,395.942,167.908,47.747,158.870
C02443=1025.153,84.955,395.923,167.910,47.743,158.869
C02444=1025.158,85.204,395.905,167.912,47.739,158.869
C02445=1025.164,85.453,395.887,167.915,47.735,158.869
C02446=1025.171,85.703,395.869,167.918,47.731,158.868
C02447=1025.176,85.952,395.851,167.920,47.728,158.868
C02448=1025.182,86.201,395.833,167.923,47.724,158.867
C02449=1025.189,86.451,395.815,167.925,47.719,158.867
C02450=1025.194,86.700,395.797,167.928,47.716,158.866
C02451=1025.200,86.949,395.779,167.931,47.712,158.866
C02452=1025.206,87.198,395.761,167.934,47.708,158.866
C02453=1025.212,87.447,395.743,167.936,47.704,158.865
C02454=1025.218,87.697,395.724,167.939,47.701,158.865
C02455=1025.224,87.946,395.706,167.941,47.696,158.864
C02456=1025.230,88.196,395.688,167.944,47.692,158.864
C02457=1025.236,88.445,395.670,167.947,47.689,158.864
C02458=1025.242,88.694,395.652,167.949,47.685,158.863
C02459=1025.248,88.943,395.633,167.951,47.680,158.863
C02460=1025.254,89.193,395.615,167.954,47.677,158.862
C02461=1025.260,89.441,395.597,167.957,47.673,158.862
C02462=1025.266,89.691,395.579,167.960,47.669,158.862
C02463=1025.272,89.940,395.560,167.961,47.666,158.861
C02464=1025.278,90.190,395.542,167.964,47.662,158.861
C02465=1025.284,90.438,395.524,167.967,47.658,158.861
C02466=1025.289,90.689,395.505,167.970,47.654,158.860
C02467=1025.296,90.938,395.487,167.972,47.651,158.860
C02468=1025.301,91.186,395.468,167.975,47.647,158.859
C02469=1025.307,91.471,395.447,167.977,47.642,158.859
C02470=1025.314,91.755,395.426,167.981,47.638,158.858
C02471=1025.321,92.039,395.405,167.984,47.634,158.858
C02472=1025.328,92.324,395.384,167.986,47.629,158.858
C02473=1025.334,92.573,395.366,167.989,47.625,158.857
C02474=1025.339,92.822,395.347,167.992,47.622,158.857
C02475=1025.345,93.072,395.329,167.995,47.618,158.856
C02476=1025.351,93.320,395.310,167.997,47.614,158.856
C02477=1025.357,93.570,395.291,167.999,47.611,158.856
C02478=1025.363,93.820,395.273,168.002,47.606,158.855
C02479=1025.370,94.069,395.255,168.005,47.602,158.855
C02480=1025.375,94.318,395.236,168.008,47.599,158.854
C02481=1025.381,94.567,395.218,168.010,47.595,158.854
C02482=1025.386,94.817,395.198,168.012,47.591,158.854
C02483=1025.392,95.065,395.180,168.015,47.587,158.853
C02484=1025.398,95.315,395.162,168.018,47.584,158.853
C02485=1025.406,95.614,395.139,168.021,47.579,158.852
C02486=1025.413,95.913,395.117,168.024,47.574,158.852
C02487=1025.420,96.213,395.095,168.027,47.570,158.851
C02488=1025.427,96.513,395.072,168.030,47.565,158.851
C02489=1025.432,96.762,395.054,168.033,47.561,158.851
C02490=1025.439,97.011,395.035,168.036,47.558,158.850
C02491=1025.445,97.260,395.016,168.038,47.553,158.850
C02492=1025.451,97.509,394.997,168.041,47.550,158.849
C02493=1025.457,97.759,394.980,168.043,47.546,158.849
C02494=1025.462,98.008,394.961,168.046,47.542,158.849
C02495=1025.469,98.257,394.942,168.049,47.538,158.848
C02496=1025.474,98.507,394.923,168.052,47.534,158.848
C02497=1025.480,98.756,394.905,168.053,47.530,158.847
C02498=1025.486,99.005,394.887,168.056,47.526,158.847
C02499=1025.492,99.254,394.867,168.059,47.523,158.847
C02500=1025.498,99.503,394.849,168.062,47.519,158.846
C02501=1025.504,99.753,394.829,168.065,47.515,158.846
C02502=1025.511,100.002,394.811,168.067,47.512,158.845
C02503=1025.516,100.251,394.792,168.070,47.508,158.845
C02504=1025.521,100.501,394.773,168.072,47.504,158.845
C02505=1025.527,100.750,394.755,168.075,47.500,158.844
C02506=1025.533,100.999,394.735,168.078,47.496,158.844
C02507=1025.539,101.249,394.716,168.080,47.493,158.843
C02508=1025.545,101.498,394.698,168.083,47.489,158.843
C02509=1025.550,101.746,394.679,168.086,47.485,158.843
C02510=1025.556,101.996,394.659,168.088,47.481,158.842
C02511=1025.562,102.245,394.641,168.090,47.477,158.842
C02512=1025.568,102.494,394.622,168.093,47.474,158.841
C02513=1025.575,102.744,394.603,168.096,47.470,158.841
C02514=1025.580,102.993,394.584,168.099,47.466,158.841
C02515=1025.585,103.242,394.565,168.102,47.462,158.840
C02516=1025.592,103.491,394.546,168.103,47.459,158.840
C02517=1025.597,103.740,394.527,168.106,47.455,158.840
C02518=1025.603,103.990,394.508,168.109,47.451,158.839
C02519=1025.610,104.239,394.489,168.112,47.447,158.839
C02520=1025.615,104.488,394.470,168.115,47.444,158.838
C02521=1025.621,104.737,394.450,168.117,47.440,158.838
C02522=1025.628,104.986,394.431,168.120,47.436,158.838
C02523=1025.633,105.235,394.412,168.123,47.433,158.837
C02524=1025.638,105.484,394.393,168.125,47.429,158.837
C02525=1025.645,105.733,394.374,168.128,47.424,158.836
C02526=1025.651,105.983,394.355,168.130,47.421,158.836
C02527=1025.656,106.232,394.336,168.133,47.417,158.836
C02528=1025.662,106.482,394.317,168.136,47.413,158.835
C02529=1025.667,106.723,394.299,168.138,47.410,158.835
C02530=1025.673,106.965,394.280,168.141,47.406,158.835
C02531=1025.679,107.207,394.261,168.143,47.402,158.834
C02532=1025.685,107.448,394.242,168.146,47.398,158.834
C02533=1025.691,107.690,394.224,168.149,47.395,158.833
C02534=1025.696,107.931,394.206,168.151,47.391,158.833
C02535=1025.703,108.173,394.187,168.154,47.387,158.833
C02536=1025.708,108.415,394.169,168.156,47.384,158.832
C02537=1025.714,108.664,394.150,168.159,47.380,158.832
C02538=1025.720,108.914,394.130,168.162,47.376,158.831
C02539=1025.726,109.162,394.111,168.164,47.373,158.831
C02540=1025.732,109.412,394.092,168.167,47.369,158.831
C02541=1025.738,109.661,394.073,168.170,47.365,158.830
C02542=1025.744,109.910,394.054,168.172,47.361,158.830
C02543=1025.750,110.160,394.035,168.175,47.357,158.829
C02544=1025.756,110.409,394.015,168.178,47.353,158.829
C02545=1025.762,110.658,393.995,168.180,47.350,158.829
C02546=1025.767,110.907,393.976,168.183,47.346,158.828
C02547=1025.773,111.156,393.957,168.186,47.342,158.828
C02548=1025.778,111.405,393.937,168.189,47.338,158.827
C02549=1025.785,111.654,393.919,168.191,47.335,158.827
C02550=1025.791,111.903,393.899,168.194,47.331,158.827
C02551=1025.797,112.152,393.879,168.196,47.327,158.826
C02552=1025.802,112.402,393.860,168.199,47.324,158.826
C02553=1025.808,112.651,393.840,168.202,47.320,158.826
C02554=1025.814,112.900,393.821,168.205,47.316,158.825
C02555=1025.820,113.149,393.802,168.208,47.312,158.825
C02556=1025.826,113.398,393.782,168.210,47.309,158.824
C02557=1025.831,113.648,393.763,168.212,47.305,158.824
C02558=1025.836,113.897,393.742,168.215,47.301,158.824
C02559=1025.842,114.146,393.723,168.218,47.297,158.823
C02560=1025.848,114.395,393.703,168.221,47.294,158.823
C02561=1025.854,114.644,393.684,168.223,47.291,158.823
C02562=1025.860,114.893,393.664,168.226,47.287,158.822
C02563=1025.866,115.143,393.644,168.229,47.283,158.822
C02564=1025.872,115.392,393.624,168.232,47.280,158.822
C02565=1025.877,115.641,393.605,168.235,47.276,158.821
C02566=1025.882,115.890,393.585,168.237,47.272,158.821
C02567=1025.888,116.140,393.565,168.239,47.269,158.820
C02568=1025.894,116.388,393.545,168.242,47.265,158.820
C02569=1025.900,116.638,393.526,168.245,47.261,158.820
C02570=1025.906,116.887,393.506,168.248,47.257,158.819
C02571=1025.912,117.136,393.487,168.250,47.254,158.819
C02572=1025.917,117.385,393.466,168.253,47.250,158.818
C02573=1025.923,117.634,393.446,168.256,47.246,158.818
C02574=1025.928,117.883,393.427,168.259,47.243,158.818
C02575=1025.934,118.132,393.407,168.261,47.239,158.817
C02576=1025.941,118.382,393.388,168.263,47.235,158.817
C02577=1025.947,118.631,393.368,168.266,47.232,158.817
C02578=1025.953,118.880,393.348,168.269,47.228,158.816
C02579=1025.958,119.130,393.328,168.272,47.224,158.816
C02580=1025.964,119.379,393.308,168.275,47.220,158.815
C02581=1025.969,119.628,393.289,168.278,47.217,158.815
C02582=1025.975,119.877,393.269,168.281,47.214,158.815
C02583=1025.981,120.126,393.249,168.283,47.210,158.814
C02584=1025.987,120.375,393.230,168.286,47.206,158.814
C02585=1025.992,120.624,393.209,168.289,47.203,158.814
C02586=1025.998,120.873,393.189,168.291,47.199,158.813
C02587=1026.004,121.122,393.170,168.294,47.195,158.813
C02588=1026.011,121.372,393.149,168.297,47.191,158.813
C02589=1026.017,121.621,393.130,168.300,47.188,158.812
C02590=1026.022,121.870,393.110,168.302,47.184,158.812
C02591=1026.028,122.119,393.090,168.305,47.180,158.811
C02592=1026.034,122.368,393.070,168.308,47.177,158.811
C02593=1026.040,122.617,393.050,168.311,47.173,158.811
C02594=1026.045,122.866,393.031,168.313,47.169,158.810
C02595=1026.051,123.115,393.011,168.316,47.165,158.810
C02596=1026.058,123.365,392.990,168.319,47.162,158.810
C02597=1026.064,123.649,392.967,168.322,47.157,158.809
C02598=1026.071,123.933,392.945,168.325,47.153,158.809
C02599=1026.078,124.217,392.922,168.328,47.149,158.808
C02600=1026.084,124.501,392.899,168.331,47.144,158.808
C02601=1026.090,124.751,392.879,168.334,47.141,158.807
C02602=1026.096,125.000,392.859,168.337,47.137,158.807
C02603=1026.102,125.249,392.840,168.340,47.133,158.807
C02604=1026.108,125.498,392.820,168.342,47.129,158.806
C02605=1026.113,125.747,392.799,168.345,47.126,158.806
C02606=1026.120,125.997,392.779,168.348,47.122,158.805
C02607=1026.126,126.246,392.759,168.351,47.118,158.805
C02608=1026.132,126.495,392.739,168.354,47.114,158.805
C02609=1026.137,126.744,392.720,168.357,47.111,158.804
C02610=1026.143,126.993,392.699,168.360,47.107,158.804
C02611=1026.149,127.242,392.679,168.363,47.103,158.804
C02612=1026.155,127.492,392.659,168.365,47.100,158.803
C02613=1026.161,127.740,392.639,168.367,47.096,158.803
C02614=1026.167,127.989,392.619,168.370,47.092,158.802
C02615=1026.174,128.239,392.599,168.373,47.089,158.802
C02616=1026.179,128.488,392.579,168.376,47.085,158.802
C02617=1026.185,128.737,392.559,168.379,47.081,158.801
C02618=1026.191,128.986,392.539,168.382,47.077,158.801
C02619=1026.197,129.235,392.518,168.384,47.073,158.800
C02620=1026.203,129.484,392.498,168.387,47.069,158.800
C02621=1026.208,129.734,392.479,168.390,47.066,158.800
C02622=1026.214,129.982,392.459,168.393,47.062,158.799
C02623=1026.221,130.232,392.438,168.396,47.058,158.799
C02624=1026.226,130.481,392.418,168.399,47.054,158.799
C02625=1026.232,130.730,392.398,168.402,47.051,158.798
C02626=1026.237,130.979,392.377,168.405,47.048,158.798
C02627=1026.244,131.228,392.356,168.407,47.044,158.797
C02628=1026.250,131.477,392.336,168.410,47.040,158.797
C02629=1026.256,131.726,392.316,168.413,47.037,158.797
C02630=1026.261,131.975,392.295,168.416,47.033,158.796
C02631=1026.267,132.224,392.275,168.418,47.029,158.796
C02632=1026.273,132.474,392.254,168.421,47.025,158.796
C02633=1026.279,132.722,392.234,168.424,47.022,158.795
C02634=1026.285,132.972,392.213,168.427,47.018,158.795
C02635=1026.291,133.221,392.193,168.430,47.015,158.795
C02636=1026.296,133.470,392.172,168.433,47.011,158.794
C02637=1026.302,133.718,392.152,168.436,47.008,158.794
C02638=1026.308,133.968,392.131,168.438,47.004,158.793
C02639=1026.314,134.217,392.111,168.441,47.000,158.793
C02640=1026.319,134.466,392.091,168.444,46.997,158.793
C02641=1026.326,134.716,392.070,168.447,46.993,158.792
C02642=1026.331,134.964,392.049,168.450,46.989,158.792
C02643=1026.337,135.213,392.029,168.453,46.985,158.792
C02644=1026.343,135.463,392.008,168.455,46.982,158.791
C02645=1026.349,135.712,391.988,168.458,46.978,158.791
C02646=1026.355,135.960,391.967,168.461,46.975,158.791
C02647=1026.361,136.210,391.946,168.464,46.971,158.790
C02648=1026.367,136.459,391.926,168.467,46.968,158.790
C02649=1026.372,136.708,391.906,168.470,46.964,158.790
C02650=1026.378,136.957,391.884,168.473,46.960,158.789
C02651=1026.384,137.206,391.864,168.476,46.956,158.789
C02652=1026.389,137.455,391.843,168.479,46.953,158.788
C02653=1026.396,137.705,391.823,168.482,46.949,158.788
C02654=1026.401,137.953,391.802,168.485,46.945,158.788
C02655=1026.407,138.203,391.781,168.488,46.942,158.787
C02656=1026.413,138.452,391.761,168.491,46.938,158.787
C02657=1026.419,138.700,391.740,168.493,46.935,158.787
C02658=1026.425,138.950,391.719,168.496,46.931,158.786
C02659=1026.430,139.199,391.698,168.498,46.928,158.786
C02660=1026.437,139.448,391.677,168.501,46.924,158.786
C02661=1026.443,139.731,391.654,168.505,46.920,158.785
C02662=1026.449,140.016,391.630,168.508,46.916,158.785
C02663=1026.456,140.300,391.606,168.512,46.912,158.784
C02664=1026.462,140.584,391.582,168.515,46.908,158.784
C02665=1026.469,140.833,391.561,168.518,46.904,158.784
C02666=1026.474,141.082,391.540,168.521,46.900,158.783
C02667=1026.480,141.332,391.520,168.524,46.897,158.783
C02668=1026.486,141.581,391.498,168.527,46.894,158.783
C02669=1026.491,141.830,391.477,168.530,46.890,158.782
C02670=1026.498,142.079,391.456,168.532,46.886,158.782
C02671=1026.503,142.328,391.436,168.535,46.883,158.782
C02672=1026.509,142.577,391.414,168.539,46.880,158.781
C02673=1026.515,142.826,391.394,168.541,46.876,158.781
C02674=1026.520,143.075,391.372,168.544,46.872,158.781
C02675=1026.527,143.324,391.351,168.547,46.868,158.780
C02676=1026.532,143.573,391.331,168.550,46.865,158.780
C02677=1026.538,143.822,391.309,168.553,46.861,158.779
C02678=1026.544,144.071,391.288,168.556,46.858,158.779
C02679=1026.550,144.320,391.267,168.559,46.854,158.779
C02680=1026.556,144.569,391.247,168.562,46.851,158.778
C02681=1026.562,144.818,391.225,168.565,46.847,158.778
C02682=1026.567,145.067,391.205,168.568,46.843,158.778
C02683=1026.573,145.317,391.183,168.571,46.839,158.777
C02684=1026.579,145.565,391.162,168.574,46.836,158.777
C02685=1026.586,145.815,391.141,168.577,46.833,158.777
C02686=1026.591,146.063,391.120,168.580,46.829,158.776
C02687=1026.597,146.312,391.099,168.583,46.825,158.776
C02688=1026.603,146.562,391.078,168.586,46.822,158.776
C02689=1026.609,146.811,391.056,168.589,46.819,158.775
C02690=1026.614,147.059,391.035,168.592,46.815,158.775
C02691=1026.620,147.309,391.014,168.595,46.811,158.775
C02692=1026.626,147.558,390.993,168.598,46.808,158.774
C02693=1026.632,147.807,390.971,168.601,46.804,158.774
C02694=1026.637,148.055,390.950,168.604,46.801,158.774
C02695=1026.643,148.305,390.929,168.607,46.797,158.773
C02696=1026.649,148.554,390.908,168.610,46.794,158.773
C02697=1026.655,148.803,390.886,168.613,46.790,158.773
C02698=1026.661,149.051,390.865,168.616,46.787,158.772
C02699=1026.667,149.301,390.843,168.618,46.783,158.772
C02700=1026.672,149.550,390.823,168.622,46.780,158.772
C02701=1026.678,149.799,390.801,168.625,46.776,158.771
C02702=1026.684,150.048,390.779,168.628,46.773,158.771
C02703=1026.689,150.297,390.758,168.631,46.770,158.771
C02704=1026.695,150.546,390.736,168.634,46.766,158.770
C02705=1026.701,150.795,390.715,168.637,46.762,158.770
C02706=1026.707,151.044,390.694,168.639,46.758,158.770
C02707=1026.712,151.293,390.673,168.643,46.755,158.769
C02708=1026.718,151.542,390.651,168.646,46.752,158.769
C02709=1026.725,151.791,390.629,168.648,46.748,158.769
C02710=1026.730,152.040,390.608,168.652,46.745,158.768
C02711=1026.736,152.289,390.586,168.655,46.741,158.768
C02712=1026.742,152.538,390.565,168.658,46.738,158.768
C02713=1026.748,152.787,390.543,168.660,46.734,158.767
C02714=1026.753,153.036,390.521,168.664,46.731,158.767
C02715=1026.759,153.285,390.500,168.667,46.727,158.767
C02716=1026.765,153.534,390.478,168.669,46.724,158.766
C02717=1026.771,153.782,390.457,168.674,46.720,158.766
C02718=1026.777,154.032,390.435,168.677,46.717,158.766
C02719=1026.783,154.281,390.414,168.680,46.713,158.765
C02720=1026.788,154.530,390.392,168.683,46.710,158.765
C02721=1026.794,154.779,390.370,168.686,46.706,158.765
C02722=1026.800,155.028,390.349,168.689,46.703,158.764
C02723=1026.806,155.277,390.327,168.692,46.700,158.764
C02724=1026.811,155.526,390.305,168.695,46.696,158.764
C02725=1026.818,155.810,390.281,168.698,46.692,158.763
C02726=1026.824,156.094,390.256,168.702,46.688,158.763
C02727=1026.831,156.377,390.231,168.705,46.684,158.763
C02728=1026.838,156.661,390.207,168.708,46.680,158.762
C02729=1026.844,156.910,390.184,168.711,46.677,158.762
C02730=1026.850,157.160,390.162,168.715,46.673,158.762
C02731=1026.855,157.408,390.141,168.718,46.670,158.762
C02732=1026.862,157.657,390.120,168.721,46.666,158.761
C02733=1026.867,157.907,390.097,168.724,46.663,158.761
C02734=1026.873,158.155,390.076,168.727,46.660,158.761
C02735=1026.879,158.404,390.054,168.730,46.656,158.760
C02736=1026.885,158.653,390.032,168.733,46.652,158.760
C02737=1026.890,158.902,390.010,168.737,46.649,158.760
C02738=1026.896,159.151,389.989,168.739,46.646,158.759
C02739=1026.902,159.400,389.967,168.742,46.642,158.759
C02740=1026.908,159.650,389.945,168.746,46.639,158.759
C02741=1026.913,159.898,389.922,168.749,46.636,158.758
C02742=1026.919,160.147,389.901,168.752,46.632,158.758
C02743=1026.925,160.396,389.878,168.755,46.629,158.758
C02744=1026.930,160.645,389.856,168.758,46.626,158.757
C02745=1026.936,160.894,389.834,168.761,46.623,158.757
C02746=1026.942,161.143,389.811,168.765,46.619,158.757
C02747=1026.946,161.392,389.789,168.768,46.616,158.757
C02748=1026.953,161.640,389.767,168.771,46.613,158.756
C02749=1026.958,161.890,389.745,168.774,46.609,158.756
C02750=1026.964,162.139,389.722,168.778,46.606,158.756
C02751=1026.969,162.388,389.700,168.780,46.602,158.755
C02752=1026.975,162.637,389.678,168.784,46.599,158.755
C02753=1026.981,162.886,389.655,168.787,46.596,158.755
C02754=1026.986,163.135,389.633,168.790,46.593,158.755
C02755=1026.992,163.383,389.611,168.793,46.590,158.754
C02756=1026.997,163.633,389.589,168.796,46.586,158.754
C02757=1027.003,163.882,389.566,168.799,46.583,158.754
C02758=1027.009,164.130,389.545,168.802,46.579,158.753
C02759=1027.014,164.379,389.522,168.805,46.576,158.753
C02760=1027.020,164.628,389.499,168.808,46.573,158.753
C02761=1027.026,164.877,389.477,168.811,46.570,158.753
C02762=1027.032,165.126,389.454,168.816,46.566,158.752
C02763=1027.037,165.375,389.432,168.819,46.563,158.752
C02764=1027.043,165.624,389.409,168.822,46.560,158.752
C02765=1027.049,165.873,389.388,168.825,46.557,158.752
C02766=1027.055,166.122,389.365,168.828,46.553,158.751
C02767=1027.060,166.371,389.343,168.831,46.550,158.751
C02768=1027.065,166.619,389.320,168.834,46.546,158.751
C02769=1027.072,166.868,389.298,168.837,46.543,158.750
C02770=1027.077,167.118,389.275,168.840,46.540,158.750
C02771=1027.083,167.366,389.252,168.844,46.536,158.750
C02772=1027.089,167.615,389.230,168.848,46.534,158.750
C02773=1027.094,167.864,389.208,168.851,46.530,158.749
C02774=1027.100,168.113,389.185,168.854,46.527,158.749
C02775=1027.105,168.362,389.162,168.857,46.523,158.749
C02776=1027.112,168.611,389.141,168.860,46.520,158.748
C02777=1027.117,168.860,389.118,168.863,46.517,158.748
C02778=1027.123,169.109,389.095,168.867,46.513,158.748
C02779=1027.129,169.358,389.073,168.870,46.510,158.748
C02780=1027.135,169.607,389.050,168.873,46.507,158.747
C02781=1027.140,169.855,389.028,168.876,46.504,158.747
C02782=1027.146,170.104,389.005,168.880,46.501,158.747
C02783=1027.152,170.353,388.983,168.883,46.497,158.746
C02784=1027.158,170.602,388.960,168.887,46.494,158.746
C02785=1027.163,170.851,388.937,168.890,46.490,158.746
C02786=1027.169,171.100,388.915,168.893,46.487,158.746
C02787=1027.175,171.349,388.893,168.896,46.483,158.745
C02788=1027.181,171.598,388.870,168.899,46.480,158.745
C02789=1027.188,171.881,388.844,168.903,46.477,158.745
C02790=1027.194,172.165,388.818,168.907,46.473,158.744
C02791=1027.201,172.448,388.792,168.911,46.469,158.744
C02792=1027.207,172.732,388.767,168.915,46.466,158.744
C02793=1027.214,172.981,388.744,168.918,46.462,158.744
C02794=1027.220,173.230,388.721,168.921,46.459,158.743
C02795=1027.225,173.479,388.698,168.924,46.455,158.743
C02796=1027.230,173.727,388.676,168.927,46.452,158.743
C02797=1027.237,173.975,388.653,168.932,46.449,158.743
C02798=1027.243,174.224,388.630,168.935,46.445,158.742
C02799=1027.248,174.474,388.608,168.938,46.442,158.742
C02800=1027.254,174.723,388.585,168.941,46.439,158.742
C02801=1027.261,174.972,388.563,168.945,46.436,158.741
C02802=1027.267,175.221,388.540,168.948,46.433,158.741
C02803=1027.272,175.470,388.517,168.951,46.429,158.741
C02804=1027.278,175.719,388.494,168.954,46.426,158.741
C02805=1027.285,175.967,388.471,168.958,46.422,158.740
C02806=1027.290,176.216,388.448,168.962,46.419,158.740
C02807=1027.296,176.465,388.425,168.965,46.416,158.740
C02808=1027.302,176.714,388.403,168.968,46.412,158.739
C02809=1027.308,176.963,388.380,168.972,46.409,158.739
C02810=1027.314,177.211,388.357,168.975,46.406,158.739
C02811=1027.320,177.460,388.334,168.978,46.403,158.739
C02812=1027.325,177.709,388.311,168.982,46.399,158.738
C02813=1027.332,177.958,388.289,168.985,46.396,158.738
C02814=1027.338,178.207,388.266,168.988,46.393,158.738
C02815=1027.343,178.456,388.243,168.993,46.389,158.738
C02816=1027.350,178.705,388.220,168.996,46.386,158.737
C02817=1027.355,178.954,388.197,168.999,46.383,158.737
C02818=1027.362,179.203,388.175,169.002,46.380,158.737
C02819=1027.368,179.452,388.152,169.006,46.376,158.736
C02820=1027.373,179.701,388.129,169.009,46.373,158.736
C02821=1027.379,179.949,388.106,169.012,46.369,158.736
C02822=1027.386,180.198,388.083,169.016,46.366,158.736
C02823=1027.391,180.447,388.060,169.020,46.363,158.735
C02824=1027.398,180.697,388.037,169.023,46.360,158.735
C02825=1027.404,180.945,388.013,169.027,46.356,158.735
C02826=1027.409,181.194,387.990,169.030,46.353,158.735
C02827=1027.416,181.442,387.968,169.033,46.350,158.734
C02828=1027.422,181.691,387.945,169.037,46.347,158.734
C02829=1027.428,181.941,387.922,169.040,46.344,158.734
C02830=1027.434,182.190,387.899,169.044,46.340,158.734
C02831=1027.440,182.438,387.876,169.048,46.337,158.733
C02832=1027.446,182.687,387.853,169.051,46.334,158.733
C02833=1027.451,182.936,387.829,169.055,46.330,158.733
C02834=1027.457,183.185,387.806,169.058,46.327,158.733
C02835=1027.464,183.434,387.782,169.061,46.324,158.732
C02836=1027.469,183.683,387.759,169.064,46.321,158.732
C02837=1027.475,183.931,387.735,169.069,46.318,158.732
C02838=1027.480,184.180,387.712,169.072,46.315,158.732
C02839=1027.486,184.429,387.688,169.075,46.312,158.731
C02840=1027.492,184.678,387.665,169.078,46.309,158.731
C02841=1027.497,184.927,387.640,169.083,46.306,158.731
C02842=1027.503,185.176,387.617,169.086,46.303,158.731
C02843=1027.508,185.424,387.593,169.089,46.300,158.731
C02844=1027.514,185.673,387.570,169.093,46.296,158.730
C02845=1027.520,185.921,387.547,169.096,46.293,158.730
C02846=1027.526,186.171,387.523,169.100,46.291,158.730
C02847=1027.532,186.420,387.499,169.103,46.288,158.730
C02848=1027.537,186.669,387.475,169.107,46.284,158.730
C02849=1027.543,186.917,387.452,169.110,46.281,158.729
C02850=1027.548,187.166,387.429,169.114,46.278,158.729
C02851=1027.554,187.415,387.404,169.118,46.275,158.729
C02852=1027.560,187.664,387.381,169.121,46.272,158.729
C02853=1027.566,187.947,387.354,169.125,46.269,158.729
C02854=1027.573,188.229,387.327,169.129,46.265,158.728
C02855=1027.580,188.513,387.300,169.134,46.262,158.728
C02856=1027.587,188.795,387.273,169.137,46.258,158.728
C02857=1027.592,189.045,387.249,169.141,46.255,158.728
C02858=1027.598,189.293,387.226,169.144,46.252,158.727
C02859=1027.604,189.542,387.202,169.148,46.249,158.727
C02860=1027.609,189.791,387.178,169.151,46.246,158.727
C02861=1027.615,190.039,387.154,169.155,46.243,158.727
C02862=1027.621,190.288,387.130,169.159,46.240,158.726
C02863=1027.627,190.537,387.106,169.162,46.237,158.726
C02864=1027.632,190.786,387.083,169.166,46.234,158.726
C02865=1027.638,191.034,387.059,169.170,46.231,158.726
C02866=1027.645,191.283,387.035,169.173,46.228,158.726
C02867=1027.650,191.532,387.011,169.177,46.225,158.726
C02868=1027.656,191.781,386.988,169.181,46.222,158.725
C02869=1027.662,192.030,386.963,169.185,46.219,158.725
C02870=1027.668,192.278,386.939,169.188,46.216,158.725
C02871=1027.674,192.527,386.916,169.191,46.213,158.725
C02872=1027.680,192.776,386.891,169.195,46.210,158.725
C02873=1027.686,193.025,386.868,169.199,46.207,158.724
C02874=1027.692,193.274,386.843,169.203,46.204,158.724
C02875=1027.698,193.523,386.820,169.206,46.201,158.724
C02876=1027.703,193.771,386.796,169.209,46.198,158.724
C02877=1027.710,194.020,386.772,169.214,46.195,158.724
C02878=1027.716,194.268,386.748,169.217,46.192,158.723
C02879=1027.721,194.518,386.724,169.221,46.189,158.723
C02880=1027.727,194.767,386.700,169.224,46.186,158.723
C02881=1027.733,195.015,386.676,169.229,46.182,158.723
C02882=1027.739,195.264,386.652,169.232,46.179,158.723
C02883=1027.744,195.513,386.628,169.236,46.176,158.722
C02884=1027.751,195.762,386.604,169.239,46.173,158.722
C02885=1027.756,196.010,386.579,169.244,46.171,158.722
C02886=1027.763,196.259,386.555,169.247,46.168,158.722
C02887=1027.769,196.508,386.532,169.251,46.165,158.722
C02888=1027.775,196.757,386.507,169.254,46.162,158.721
C02889=1027.781,197.005,386.484,169.258,46.159,158.721
C02890=1027.787,197.254,386.459,169.262,46.156,158.721
C02891=1027.793,197.503,386.435,169.265,46.153,158.721
C02892=1027.799,197.752,386.411,169.269,46.149,158.721
C02893=1027.805,198.000,386.387,169.273,46.146,158.720
C02894=1027.811,198.250,386.362,169.277,46.143,158.720
C02895=1027.817,198.498,386.339,169.281,46.141,158.720
C02896=1027.823,198.747,386.314,169.285,46.138,158.720
C02897=1027.829,198.995,386.290,169.289,46.135,158.720
C02898=1027.835,199.244,386.266,169.292,46.132,158.720
C02899=1027.841,199.493,386.242,169.296,46.128,158.719
C02900=1027.847,199.742,386.218,169.300,46.126,158.719
C02901=1027.853,199.990,386.193,169.304,46.122,158.719
C02902=1027.860,200.239,386.169,169.307,46.119,158.719
C02903=1027.865,200.488,386.144,169.312,46.117,158.719
C02904=1027.871,200.737,386.120,169.315,46.114,158.719
C02905=1027.877,200.986,386.096,169.319,46.111,158.718
C02906=1027.882,201.234,386.071,169.323,46.108,158.718
C02907=1027.889,201.483,386.047,169.327,46.105,158.718
C02908=1027.894,201.732,386.022,169.330,46.102,158.718
C02909=1027.900,201.980,385.997,169.335,46.100,158.718
C02910=1027.906,202.229,385.973,169.338,46.097,158.718
C02911=1027.912,202.478,385.948,169.342,46.094,158.717
C02912=1027.918,202.727,385.923,169.346,46.091,158.717
C02913=1027.924,202.975,385.899,169.350,46.088,158.717
C02914=1027.930,203.224,385.874,169.353,46.085,158.717
C02915=1027.935,203.472,385.850,169.358,46.083,158.717
C02916=1027.941,203.722,385.825,169.361,46.080,158.717
C02917=1027.966,204.765,385.721,169.737,46.183,158.781
C02918=1027.977,205.147,385.681,169.742,46.180,158.781
C02919=1027.987,205.530,385.641,169.746,46.176,158.781
C02920=1027.998,205.912,385.601,169.750,46.173,158.781
C02921=1028.008,206.294,385.561,169.755,46.170,158.780
C02922=1028.015,206.542,385.535,169.757,46.169,158.781
C02923=1028.021,206.791,385.508,169.761,46.166,158.780
C02924=1028.027,207.040,385.482,169.763,46.164,158.780
C02925=1028.034,207.289,385.456,169.766,46.162,158.780
C02926=1028.041,207.537,385.430,169.769,46.160,158.780
C02927=1028.048,207.786,385.404,169.772,46.158,158.780
C02928=1028.054,208.034,385.378,169.775,46.157,158.780
C02929=1028.061,208.283,385.351,169.778,46.154,158.780
C02930=1028.067,208.531,385.324,169.781,46.152,158.780
C02931=1028.074,208.780,385.298,169.784,46.150,158.780
C02932=1028.081,209.028,385.272,169.786,46.148,158.779
C02933=1028.087,209.277,385.245,169.789,46.147,158.779
C02934=1028.093,209.525,385.220,169.793,46.144,158.779
C02935=1028.101,209.774,385.193,169.795,46.142,158.779
C02936=1028.107,210.022,385.167,169.798,46.140,158.779
C02937=1028.113,210.271,385.140,169.801,46.139,158.779
C02938=1028.120,210.519,385.114,169.804,46.137,158.779
C02939=1028.127,210.768,385.088,169.806,46.135,158.779
C02940=1028.133,211.016,385.061,169.810,46.132,158.779
C02941=1028.140,211.265,385.035,169.813,46.131,158.779
C02942=1028.147,211.513,385.008,169.815,46.129,158.779
C02943=1028.153,211.762,384.981,169.819,46.127,158.779
C02944=1028.160,212.010,384.954,169.821,46.125,158.779
C02945=1028.166,212.259,384.928,169.824,46.123,158.778
C02946=1028.173,212.508,384.901,169.827,46.121,158.778
C02947=1028.179,212.756,384.875,169.830,46.119,158.778
C02948=1028.186,213.005,384.848,169.833,46.117,158.778
C02949=1028.193,213.253,384.822,169.836,46.115,158.778
C02950=1028.199,213.502,384.795,169.839,46.114,158.778
C02951=1028.206,213.750,384.768,169.842,46.111,158.778
C02952=1028.212,213.998,384.741,169.845,46.110,158.778
C02953=1028.219,214.247,384.715,169.848,46.108,158.778
C02954=1028.225,214.495,384.688,169.851,46.106,158.778
C02955=1028.232,214.744,384.662,169.854,46.104,158.778
C02956=1028.239,214.993,384.636,169.856,46.102,158.778
C02957=1028.245,215.241,384.608,169.860,46.100,158.778
C02958=1028.252,215.489,384.582,169.863,46.099,158.778
C02959=1028.258,215.738,384.555,169.865,46.097,158.778
C02960=1028.265,215.986,384.529,169.869,46.095,158.778
C02961=1028.272,216.235,384.501,169.871,46.093,158.777
C02962=1028.279,216.483,384.475,169.875,46.091,158.777
C02963=1028.285,216.732,384.448,169.878,46.089,158.777
C02964=1028.292,216.981,384.421,169.880,46.087,158.777
C02965=1028.299,217.228,384.395,169.884,46.086,158.777
C02966=1028.305,217.477,384.368,169.886,46.084,158.777
C02967=1028.312,217.726,384.341,169.890,46.081,158.777
C02968=1028.318,217.974,384.315,169.893,46.080,158.777
C02969=1028.326,218.222,384.287,169.895,46.078,158.777
C02970=1028.332,218.472,384.260,169.899,46.076,158.777
C02971=1028.338,218.720,384.234,169.901,46.074,158.777
C02972=1028.345,218.968,384.207,169.905,46.073,158.777
C02973=1028.352,219.217,384.180,169.908,46.071,158.777
C02974=1028.362,219.604,384.138,169.912,46.068,158.777
C02975=1028.372,219.991,384.096,169.918,46.065,158.777
C02976=1028.382,220.378,384.054,169.922,46.062,158.777
C02977=1028.393,220.766,384.012,169.926,46.060,158.777
C02978=1028.399,221.014,383.984,169.929,46.058,158.777
C02979=1028.406,221.263,383.957,169.933,46.056,158.777
C02980=1028.412,221.511,383.930,169.935,46.055,158.777
C02981=1028.419,221.759,383.904,169.939,46.053,158.777
C02982=1028.426,222.008,383.876,169.942,46.051,158.776
C02983=1028.432,222.256,383.848,169.944,46.050,158.776
C02984=1028.439,222.505,383.821,169.948,46.047,158.776
C02985=1028.445,222.753,383.794,169.951,46.046,158.776
C02986=1028.452,223.002,383.767,169.954,46.044,158.776
C02987=1028.459,223.250,383.740,169.957,46.042,158.776
C02988=1028.465,223.499,383.713,169.960,46.041,158.776
C02989=1028.472,223.747,383.686,169.963,46.039,158.776
C02990=1028.478,223.995,383.658,169.966,46.037,158.776
C02991=1028.485,224.244,383.631,169.970,46.036,158.776
C02992=1028.492,224.492,383.604,169.972,46.034,158.776
C02993=1028.498,224.740,383.577,169.975,46.032,158.776
C02994=1028.505,224.989,383.550,169.979,46.031,158.776
C02995=1028.511,225.238,383.522,169.981,46.029,158.776
C02996=1028.518,225.486,383.496,169.985,46.027,158.776
C02997=1028.525,225.735,383.468,169.987,46.025,158.776
C02998=1028.532,225.983,383.440,169.991,46.023,158.776
C02999=1028.538,226.231,383.413,169.994,46.022,158.776
C03000=1028.545,226.480,383.386,169.996,46.020,158.776
C03001=1028.552,226.728,383.359,170.000,46.018,158.776
C03002=1028.558,226.977,383.331,170.003,46.017,158.776
C03003=1028.565,227.226,383.304,170.006,46.015,158.776
C03004=1028.572,227.474,383.277,170.009,46.013,158.776
C03005=1028.578,227.721,383.249,170.013,46.012,158.776
C03006=1028.585,227.970,383.222,170.016,46.010,158.776
C03007=1028.592,228.218,383.194,170.018,46.009,158.776
C03008=1028.598,228.467,383.166,170.022,46.007,158.776
C03009=1028.605,228.716,383.139,170.025,46.005,158.776
C03010=1028.611,228.964,383.111,170.028,46.004,158.776
C03011=1028.617,229.212,383.084,170.031,46.002,158.776
C03012=1028.624,229.460,383.056,170.035,46.001,158.776
C03013=1028.631,229.709,383.029,170.037,45.999,158.776
C03014=1028.637,229.957,383.001,170.040,45.997,158.776
C03015=1028.644,230.206,382.973,170.044,45.996,158.776
C03016=1028.651,230.454,382.945,170.047,45.994,158.776
C03017=1028.657,230.703,382.918,170.051,45.993,158.776
C03018=1028.664,230.951,382.890,170.053,45.990,158.776
C03019=1028.670,231.199,382.863,170.057,45.989,158.776
C03020=1028.677,231.447,382.835,170.060,45.987,158.776
C03021=1028.683,231.696,382.806,170.062,45.986,158.776
C03022=1028.690,231.944,382.779,170.066,45.984,158.776
C03023=1028.696,232.193,382.751,170.069,45.983,158.776
C03024=1028.703,232.441,382.723,170.073,45.981,158.776
C03025=1028.710,232.690,382.696,170.075,45.980,158.776
C03026=1028.716,232.938,382.668,170.079,45.978,158.776
C03027=1028.723,233.187,382.640,170.082,45.977,158.776
C03028=1028.729,233.435,382.612,170.085,45.976,158.776
C03029=1028.735,233.683,382.584,170.088,45.974,158.777
C03030=1028.746,234.062,382.542,170.093,45.972,158.776
C03031=1028.756,234.442,382.499,170.097,45.969,158.776
C03032=1028.766,234.822,382.456,170.103,45.967,158.777
C03033=1028.776,235.202,382.413,170.108,45.964,158.777
C03034=1028.783,235.450,382.386,170.111,45.963,158.777
C03035=1028.789,235.699,382.358,170.114,45.961,158.777
C03036=1028.796,235.946,382.330,170.117,45.960,158.777
C03037=1028.803,236.195,382.302,170.121,45.958,158.777
C03038=1028.809,236.444,382.273,170.124,45.957,158.777
C03039=1028.815,236.692,382.246,170.127,45.956,158.777
C03040=1028.822,236.941,382.218,170.130,45.954,158.777
C03041=1028.829,237.188,382.190,170.134,45.953,158.777
C03042=1028.836,237.437,382.162,170.137,45.951,158.777
C03043=1028.843,237.685,382.134,170.140,45.950,158.777
C03044=1028.849,237.933,382.105,170.143,45.948,158.777
C03045=1028.855,238.182,382.077,170.147,45.947,158.777
C03046=1028.862,238.430,382.050,170.150,45.945,158.777
C03047=1028.869,238.678,382.021,170.153,45.944,158.777
C03048=1028.875,238.927,381.993,170.156,45.942,158.777
C03049=1028.882,239.175,381.965,170.160,45.941,158.777
C03050=1028.889,239.423,381.937,170.163,45.939,158.777
C03051=1028.895,239.672,381.909,170.167,45.938,158.778
C03052=1028.902,239.920,381.881,170.170,45.937,158.778
C03053=1028.908,240.168,381.852,170.173,45.935,158.778
C03054=1028.915,240.417,381.824,170.176,45.934,158.778
C03055=1028.921,240.665,381.795,170.180,45.932,158.778
C03056=1028.928,240.913,381.768,170.183,45.931,158.778
C03057=1028.934,241.161,381.739,170.186,45.929,158.778
C03058=1028.941,241.410,381.711,170.189,45.928,158.778
C03059=1028.948,241.659,381.681,170.192,45.927,158.778
C03060=1028.954,241.907,381.654,170.196,45.925,158.778
C03061=1028.961,242.155,381.625,170.199,45.924,158.778
C03062=1028.968,242.403,381.596,170.203,45.923,158.778
C03063=1028.974,242.652,381.568,170.206,45.922,158.778
C03064=1028.981,242.899,381.539,170.209,45.920,158.778
C03065=1028.987,243.148,381.511,170.212,45.919,158.778
C03066=1028.994,243.396,381.483,170.216,45.917,158.778
C03067=1029.000,243.644,381.454,170.219,45.916,158.779
C03068=1029.007,243.893,381.426,170.223,45.915,158.779
C03069=1029.014,244.141,381.397,170.225,45.913,158.779
C03070=1029.020,244.390,381.369,170.229,45.912,158.779
C03071=1029.026,244.638,381.340,170.232,45.911,158.779
C03072=1029.032,244.886,381.311,170.236,45.909,158.779
C03073=1029.039,245.134,381.282,170.239,45.909,158.779
C03074=1029.046,245.382,381.253,170.243,45.907,158.779
C03075=1029.052,245.631,381.225,170.246,45.906,158.779
C03076=1029.058,245.879,381.196,170.250,45.905,158.780
C03077=1029.065,246.128,381.167,170.252,45.903,158.780
C03078=1029.072,246.376,381.138,170.256,45.902,158.780
C03079=1029.078,246.624,381.109,170.259,45.901,158.780
C03080=1029.084,246.873,381.081,170.263,45.899,158.780
C03081=1029.091,247.120,381.052,170.266,45.899,158.780
C03082=1029.097,247.368,381.023,170.270,45.897,158.780
C03083=1029.104,247.617,380.994,170.273,45.896,158.780
C03084=1029.110,247.865,380.965,170.277,45.895,158.780
C03085=1029.117,248.114,380.936,170.280,45.894,158.781
C03086=1029.127,248.487,380.892,170.285,45.892,158.781
C03087=1029.136,248.861,380.849,170.290,45.890,158.781
C03088=1029.146,249.234,380.806,170.295,45.888,158.781
C03089=1029.156,249.608,380.762,170.300,45.886,158.781
C03090=1029.162,249.856,380.733,170.304,45.885,158.781
C03091=1029.169,250.104,380.704,170.307,45.884,158.781
C03092=1029.176,250.352,380.675,170.311,45.883,158.782
C03093=1029.182,250.601,380.646,170.314,45.881,158.782
C03094=1029.189,250.849,380.617,170.317,45.881,158.782
C03095=1029.196,251.097,380.588,170.321,45.879,158.782
C03096=1029.203,251.346,380.559,170.324,45.878,158.782
C03097=1029.209,251.594,380.530,170.328,45.877,158.782
C03098=1029.215,251.842,380.501,170.331,45.876,158.782
C03099=1029.221,252.090,380.472,170.335,45.874,158.782
C03100=1029.229,252.338,380.443,170.338,45.874,158.783
C03101=1029.235,252.587,380.414,170.342,45.872,158.783
C03102=1029.242,252.834,380.384,170.346,45.871,158.783
C03103=1029.249,253.083,380.355,170.348,45.870,158.783
C03104=1029.255,253.331,380.326,170.352,45.869,158.783
C03105=1029.262,253.579,380.297,170.355,45.867,158.783
C03106=1029.269,253.828,380.268,170.359,45.866,158.783
C03107=1029.275,254.076,380.239,170.362,45.865,158.783
C03108=1029.281,254.324,380.210,170.366,45.864,158.784
C03109=1029.289,254.572,380.180,170.370,45.863,158.784
C03110=1029.295,254.820,380.151,170.373,45.862,158.784
C03111=1029.302,255.069,380.122,170.377,45.861,158.784
C03112=1029.308,255.317,380.093,170.380,45.859,158.784
C03113=1029.315,255.565,380.064,170.384,45.858,158.784
C03114=1029.322,255.813,380.034,170.387,45.857,158.784
C03115=1029.329,256.061,380.005,170.390,45.856,158.785
C03116=1029.336,256.310,379.976,170.395,45.855,158.785
C03117=1029.342,256.558,379.947,170.397,45.854,158.785
C03118=1029.348,256.806,379.917,170.401,45.853,158.785
C03119=1029.356,257.054,379.888,170.405,45.852,158.785
C03120=1029.362,257.302,379.859,170.408,45.850,158.785
C03121=1029.369,257.550,379.829,170.412,45.849,158.786
C03122=1029.376,257.799,379.800,170.416,45.848,158.786
C03123=1029.382,258.047,379.771,170.419,45.847,158.786
C03124=1029.389,258.295,379.741,170.423,45.846,158.786
C03125=1029.397,258.543,379.712,170.426,45.845,158.786
C03126=1029.403,258.792,379.683,170.430,45.844,158.786
C03127=1029.410,259.040,379.653,170.434,45.843,158.787
C03128=1029.416,259.288,379.624,170.437,45.841,158.787
C03129=1029.423,259.537,379.594,170.441,45.841,158.787
C03130=1029.430,259.784,379.565,170.445,45.840,158.787
C03131=1029.437,260.033,379.536,170.447,45.838,158.787
C03132=1029.444,260.280,379.506,170.452,45.837,158.787
C03133=1029.451,260.529,379.477,170.456,45.836,158.787
C03134=1029.457,260.777,379.447,170.458,45.835,158.787
C03135=1029.465,261.025,379.418,170.462,45.834,158.788
C03136=1029.471,261.273,379.388,170.466,45.833,158.788
C03137=1029.477,261.522,379.358,170.469,45.832,158.788
C03138=1029.484,261.769,379.329,170.473,45.831,158.788
C03139=1029.491,262.018,379.298,170.478,45.830,158.789
C03140=1029.497,262.266,379.269,170.480,45.829,158.789
C03141=1029.504,262.514,379.239,170.484,45.828,158.789
C03142=1029.514,262.886,379.194,170.489,45.827,158.789
C03143=1029.524,263.258,379.150,170.495,45.825,158.789
C03144=1029.534,263.630,379.105,170.501,45.824,158.790
C03145=1029.543,264.002,379.060,170.507,45.823,158.790
C03146=1029.550,264.250,379.030,170.510,45.822,158.790
C03147=1029.557,264.498,379.000,170.514,45.821,158.791
C03148=1029.564,264.746,378.970,170.518,45.820,158.791
C03149=1029.570,264.995,378.940,170.521,45.819,158.791
C03150=1029.577,265.242,378.910,170.525,45.818,158.791
C03151=1029.584,265.491,378.880,170.528,45.817,158.791
C03152=1029.590,265.739,378.851,170.532,45.817,158.792
C03153=1029.597,265.987,378.821,170.536,45.815,158.792
C03154=1029.604,266.235,378.790,170.540,45.814,158.792
C03155=1029.610,266.483,378.760,170.543,45.813,158.792
C03156=1029.618,266.731,378.730,170.547,45.813,158.792
C03157=1029.623,266.979,378.700,170.550,45.812,158.793
C03158=1029.631,267.227,378.669,170.554,45.811,158.793
C03159=1029.638,267.475,378.639,170.558,45.810,158.793
C03160=1029.644,267.723,378.609,170.562,45.809,158.793
C03161=1029.651,267.971,378.579,170.565,45.809,158.793
C03162=1029.657,268.220,378.548,170.569,45.808,158.794
C03163=1029.664,268.467,378.518,170.573,45.807,158.794
C03164=1029.671,268.716,378.488,170.576,45.806,158.794
C03165=1029.677,268.964,378.458,170.580,45.805,158.794
C03166=1029.684,269.212,378.428,170.584,45.804,158.795
C03167=1029.691,269.460,378.398,170.587,45.803,158.795
C03168=1029.697,269.708,378.367,170.592,45.803,158.795
C03169=1029.704,269.956,378.337,170.596,45.802,158.795
C03170=1029.710,270.204,378.306,170.599,45.801,158.796
C03171=1029.718,270.453,378.276,170.603,45.800,158.796
C03172=1029.723,270.700,378.246,170.607,45.799,158.796
C03173=1029.731,270.948,378.215,170.610,45.798,158.796
C03174=1029.737,271.196,378.184,170.614,45.798,158.797
C03175=1029.744,271.444,378.155,170.618,45.797,158.797
C03176=1029.750,271.693,378.124,170.622,45.796,158.797
C03177=1029.757,271.941,378.094,170.625,45.795,158.797
C03178=1029.764,272.189,378.062,170.630,45.795,158.798
C03179=1029.771,272.436,378.033,170.634,45.794,158.798
C03180=1029.777,272.685,378.002,170.637,45.793,158.798
C03181=1029.784,272.932,377.971,170.641,45.792,158.798
C03182=1029.791,273.181,377.940,170.645,45.792,158.799
C03183=1029.797,273.429,377.910,170.649,45.791,158.799
C03184=1029.804,273.677,377.880,170.652,45.790,158.799
C03185=1029.811,273.925,377.848,170.657,45.790,158.799
C03186=1029.818,274.173,377.818,170.661,45.789,158.800
C03187=1029.824,274.420,377.787,170.664,45.788,158.800
C03188=1029.830,274.669,377.757,170.668,45.788,158.800
C03189=1029.837,274.917,377.726,170.672,45.787,158.800
C03190=1029.844,275.165,377.695,170.676,45.786,158.801
C03191=1029.851,275.413,377.664,170.679,45.786,158.801
C03192=1029.857,275.660,377.634,170.683,45.785,158.801
C03193=1029.864,275.909,377.603,170.687,45.784,158.802
C03194=1029.871,276.157,377.572,170.692,45.784,158.802
C03195=1029.878,276.405,377.542,170.695,45.783,158.802
C03196=1029.885,276.653,377.510,170.699,45.783,158.802
C03197=1029.891,276.901,377.479,170.703,45.782,158.803
C03198=1029.901,277.277,377.432,170.709,45.781,158.803
C03199=1029.912,277.654,377.386,170.714,45.780,158.804
C03200=1029.922,278.031,377.339,170.721,45.779,158.804
C03201=1029.932,278.407,377.292,170.727,45.778,158.805
C03202=1029.938,278.656,377.261,170.730,45.777,158.805
C03203=1029.945,278.903,377.229,170.735,45.777,158.805
C03204=1029.952,279.151,377.198,170.739,45.777,158.806
C03205=1029.958,279.399,377.167,170.743,45.776,158.806
C03206=1029.965,279.648,377.136,170.747,45.775,158.806
C03207=1029.972,279.895,377.105,170.750,45.775,158.806
C03208=1029.979,280.143,377.074,170.755,45.774,158.807
C03209=1029.986,280.391,377.042,170.759,45.773,158.807
C03210=1029.992,280.640,377.011,170.763,45.773,158.807
C03211=1029.998,280.887,376.980,170.766,45.773,158.808
C03212=1030.005,281.135,376.949,170.770,45.772,158.808
C03213=1030.012,281.383,376.918,170.775,45.772,158.808
C03214=1030.018,281.631,376.886,170.779,45.771,158.809
C03215=1030.025,281.879,376.855,170.783,45.770,158.809
C03216=1030.031,282.127,376.824,170.786,45.770,158.809
C03217=1030.039,282.375,376.793,170.790,45.769,158.809
C03218=1030.046,282.623,376.762,170.795,45.769,158.810
C03219=1030.052,282.870,376.730,170.799,45.768,158.810
C03220=1030.059,283.118,376.699,170.803,45.767,158.811
C03221=1030.066,283.366,376.667,170.806,45.767,158.811
C03222=1030.073,283.614,376.636,170.811,45.767,158.811
C03223=1030.079,283.862,376.605,170.815,45.767,158.812
C03224=1030.086,284.110,376.573,170.819,45.766,158.812
C03225=1030.093,284.358,376.542,170.823,45.765,158.812
C03226=1030.099,284.606,376.510,170.828,45.765,158.813
C03227=1030.106,284.854,376.479,170.831,45.764,158.813
C03228=1030.114,285.101,376.448,170.835,45.764,158.813
C03229=1030.121,285.350,376.416,170.839,45.764,158.814
C03230=1030.128,285.598,376.385,170.844,45.763,158.814
C03231=1030.134,285.846,376.353,170.848,45.762,158.814
C03232=1030.141,286.094,376.322,170.852,45.762,158.815
C03233=1030.148,286.341,376.290,170.856,45.762,158.815
C03234=1030.155,286.589,376.258,170.859,45.762,158.815
C03235=1030.161,286.837,376.226,170.864,45.761,158.816
C03236=1030.168,287.085,376.195,170.868,45.761,158.816
C03237=1030.174,287.333,376.163,170.872,45.760,158.816
C03238=1030.181,287.580,376.131,170.876,45.760,158.817
C03239=1030.188,287.828,376.100,170.881,45.759,158.817
C03240=1030.195,288.076,376.068,170.885,45.759,158.818
C03241=1030.202,288.324,376.037,170.888,45.759,158.818
C03242=1030.209,288.572,376.004,170.893,45.758,158.818
C03243=1030.215,288.820,375.972,170.897,45.758,158.819
C03244=1030.222,289.068,375.941,170.901,45.758,158.819
C03245=1030.229,289.315,375.909,170.906,45.757,158.820
C03246=1030.236,289.563,375.877,170.910,45.757,158.820
C03247=1030.243,289.810,375.845,170.914,45.757,158.820
C03248=1030.249,290.059,375.813,170.918,45.757,158.821
C03249=1030.256,290.307,375.781,170.922,45.756,158.821
C03250=1030.263,290.554,375.749,170.926,45.756,158.821
C03251=1030.270,290.802,375.718,170.931,45.756,158.822
C03252=1030.276,291.050,375.685,170.935,45.755,158.822
C03253=1030.283,291.299,375.653,170.939,45.755,158.823
C03254=1030.293,291.687,375.603,170.946,45.755,158.823
C03255=1030.305,292.076,375.553,170.952,45.754,158.824
C03256=1030.316,292.465,375.502,170.959,45.754,158.825
C03257=1030.326,292.854,375.452,170.966,45.753,158.825
C03258=1030.333,293.101,375.420,170.970,45.753,158.826
C03259=1030.340,293.349,375.387,170.974,45.753,158.826
C03260=1030.347,293.597,375.356,170.978,45.752,158.826
C03261=1030.354,293.844,375.324,170.983,45.752,158.827
C03262=1030.361,294.093,375.291,170.987,45.752,158.827
C03263=1030.367,294.341,375.259,170.991,45.752,158.828
C03264=1030.374,294.588,375.226,170.996,45.752,158.828
C03265=1030.381,294.835,375.194,171.000,45.751,158.829
C03266=1030.387,295.084,375.161,171.005,45.752,158.829
C03267=1030.394,295.331,375.128,171.009,45.751,158.829
C03268=1030.400,295.579,375.097,171.013,45.751,158.830
C03269=1030.407,295.827,375.064,171.017,45.751,158.830
C03270=1030.414,296.075,375.031,171.021,45.751,158.831
C03271=1030.421,296.322,374.999,171.026,45.751,158.831
C03272=1030.427,296.570,374.966,171.030,45.751,158.832
C03273=1030.434,296.818,374.933,171.034,45.751,158.832
C03274=1030.441,297.066,374.901,171.039,45.750,158.833
C03275=1030.447,297.313,374.868,171.043,45.751,158.833
C03276=1030.453,297.561,374.835,171.048,45.750,158.833
C03277=1030.461,297.809,374.803,171.052,45.751,158.834
C03278=1030.467,298.056,374.770,171.057,45.750,158.834
C03279=1030.474,298.304,374.737,171.061,45.750,158.835
C03280=1030.481,298.552,374.705,171.065,45.750,158.835
C03281=1030.488,298.800,374.672,171.070,45.750,158.836
C03282=1030.495,299.048,374.639,171.074,45.750,158.836
C03283=1030.501,299.295,374.606,171.079,45.750,158.837
C03284=1030.508,299.542,374.573,171.083,45.750,158.837
C03285=1030.515,299.790,374.540,171.088,45.750,158.838
C03286=1030.521,300.038,374.508,171.092,45.750,158.838
C03287=1030.529,300.286,374.475,171.096,45.750,158.839
C03288=1030.535,300.534,374.442,171.101,45.750,158.839
C03289=1030.542,300.782,374.409,171.105,45.749,158.840
C03290=1030.550,301.028,374.376,171.110,45.750,158.840
C03291=1030.556,301.276,374.344,171.115,45.750,158.841
C03292=1030.563,301.524,374.311,171.119,45.750,158.841
C03293=1030.569,301.772,374.278,171.123,45.750,158.842
C03294=1030.577,302.019,374.245,171.128,45.750,158.842
C03295=1030.583,302.267,374.212,171.132,45.750,158.843
C03296=1030.590,302.515,374.179,171.137,45.750,158.843
C03297=1030.597,302.762,374.147,171.141,45.750,158.844
C03298=1030.604,303.010,374.113,171.146,45.750,158.844
C03299=1030.611,303.258,374.080,171.150,45.750,158.845
C03300=1030.618,303.506,374.047,171.155,45.750,158.845
C03301=1030.625,303.753,374.014,171.159,45.750,158.846
C03302=1030.632,304.001,373.981,171.164,45.750,158.846
C03303=1030.639,304.249,373.947,171.168,45.750,158.847
C03304=1030.645,304.496,373.914,171.173,45.750,158.847
C03305=1030.653,304.744,373.882,171.177,45.750,158.848
C03306=1030.660,304.992,373.848,171.182,45.750,158.848
C03307=1030.666,305.240,373.815,171.186,45.750,158.849
C03308=1030.674,305.487,373.782,171.191,45.750,158.849
C03309=1030.681,305.734,373.749,171.195,45.751,158.850
C03310=1030.692,306.140,373.695,171.203,45.751,158.851
C03311=1030.704,306.546,373.640,171.211,45.751,158.852
C03312=1030.716,306.952,373.585,171.219,45.750,158.852
C03313=1030.727,307.359,373.531,171.225,45.751,158.853
C03314=1030.734,307.606,373.498,171.230,45.751,158.854
C03315=1030.741,307.853,373.464,171.236,45.751,158.854
C03316=1030.749,308.101,373.432,171.240,45.751,158.855
C03317=1030.756,308.349,373.398,171.245,45.752,158.855
C03318=1030.763,308.596,373.364,171.249,45.751,158.856
C03319=1030.769,308.844,373.331,171.254,45.752,158.856
C03320=1030.777,309.092,373.298,171.258,45.752,158.857
C03321=1030.785,309.339,373.264,171.263,45.752,158.858
C03322=1030.791,309.587,373.231,171.268,45.752,158.858
C03323=1030.798,309.835,373.198,171.273,45.752,158.859
C03324=1030.805,310.082,373.164,171.278,45.753,158.859
C03325=1030.813,310.330,373.130,171.282,45.752,158.860
C03326=1030.820,310.577,373.097,171.287,45.753,158.860
C03327=1030.827,310.825,373.064,171.291,45.753,158.861
C03328=1030.834,311.073,373.030,171.297,45.753,158.861
C03329=1030.841,311.320,372.996,171.301,45.753,158.862
C03330=1030.848,311.568,372.962,171.306,45.753,158.863
C03331=1030.855,311.815,372.929,171.311,45.754,158.863
C03332=1030.861,312.063,372.895,171.315,45.755,158.864
C03333=1030.869,312.310,372.860,171.320,45.755,158.864
C03334=1030.876,312.558,372.826,171.325,45.755,158.865
C03335=1030.882,312.805,372.792,171.329,45.755,158.866
C03336=1030.889,313.053,372.758,171.335,45.756,158.866
C03337=1030.896,313.300,372.725,171.340,45.756,158.867
C03338=1030.903,313.548,372.690,171.344,45.757,158.867
C03339=1030.910,313.795,372.656,171.349,45.757,158.868
C03340=1030.917,314.043,372.622,171.354,45.758,158.869
C03341=1030.923,314.290,372.588,171.358,45.758,158.869
C03342=1030.931,314.538,372.554,171.363,45.758,158.870
C03343=1030.937,314.785,372.519,171.368,45.758,158.871
C03344=1030.945,315.033,372.485,171.373,45.759,158.871
C03345=1030.952,315.281,372.451,171.378,45.759,158.872
C03346=1030.958,315.529,372.417,171.382,45.760,158.872
C03347=1030.966,315.776,372.382,171.387,45.761,158.873
C03348=1030.973,316.023,372.348,171.393,45.761,158.874
C03349=1030.979,316.271,372.314,171.398,45.761,158.875
C03350=1030.986,316.518,372.280,171.402,45.762,158.875
C03351=1030.993,316.766,372.245,171.407,45.762,158.876
C03352=1031.000,317.013,372.211,171.412,45.763,158.876
C03353=1031.007,317.260,372.177,171.417,45.763,158.877
C03354=1031.014,317.508,372.142,171.422,45.763,158.878
C03355=1031.021,317.756,372.108,171.427,45.764,158.878
C03356=1031.028,318.003,372.073,171.431,45.764,158.879
C03357=1031.035,318.251,372.039,171.436,45.765,158.880
C03358=1031.043,318.498,372.004,171.442,45.765,158.880
C03359=1031.049,318.746,371.970,171.447,45.766,158.881
C03360=1031.057,318.993,371.935,171.451,45.766,158.882
C03361=1031.064,319.241,371.901,171.456,45.767,158.882
C03362=1031.071,319.488,371.866,171.462,45.767,158.883
C03363=1031.079,319.736,371.832,171.467,45.768,158.884
C03364=1031.085,319.983,371.797,171.471,45.768,158.884
C03365=1031.093,320.230,371.763,171.477,45.769,158.885
C03366=1031.105,320.642,371.706,171.485,45.770,158.886
C03367=1031.116,321.053,371.649,171.493,45.770,158.887
C03368=1031.129,321.464,371.591,171.502,45.772,158.888
C03369=1031.140,321.874,371.532,171.510,45.773,158.889
C03370=1031.148,322.122,371.498,171.515,45.773,158.890
C03371=1031.155,322.369,371.464,171.521,45.773,158.891
C03372=1031.162,322.616,371.429,171.525,45.774,158.892
C03373=1031.169,322.863,371.394,171.530,45.775,158.892
C03374=1031.176,323.112,371.359,171.536,45.775,158.893
C03375=1031.184,323.359,371.325,171.541,45.776,158.894
C03376=1031.191,323.607,371.290,171.546,45.777,158.894
C03377=1031.198,323.854,371.255,171.551,45.777,158.895
C03378=1031.206,324.101,371.220,171.556,45.778,158.896
C03379=1031.213,324.349,371.185,171.561,45.779,158.896
C03380=1031.221,324.596,371.151,171.567,45.779,158.897
C03381=1031.228,324.844,371.115,171.571,45.780,158.898
C03382=1031.235,325.091,371.081,171.577,45.780,158.899
C03383=1031.242,325.338,371.045,171.582,45.781,158.899
C03384=1031.250,325.586,371.010,171.587,45.782,158.900
C03385=1031.257,325.833,370.975,171.593,45.783,158.901
C03386=1031.265,326.080,370.941,171.597,45.783,158.901
C03387=1031.273,326.328,370.906,171.603,45.783,158.902
C03388=1031.280,326.576,370.871,171.608,45.784,158.903
C03389=1031.288,326.823,370.836,171.613,45.785,158.904
C03390=1031.294,327.071,370.801,171.619,45.786,158.905
C03391=1031.302,327.318,370.766,171.624,45.787,158.905
C03392=1031.309,327.566,370.731,171.630,45.787,158.906
C03393=1031.317,327.813,370.696,171.634,45.787,158.907
C03394=1031.324,328.060,370.660,171.640,45.788,158.907
C03395=1031.331,328.308,370.625,171.645,45.790,158.908
C03396=1031.338,328.555,370.590,171.650,45.790,158.909
C03397=1031.346,328.802,370.553,171.656,45.791,158.910
C03398=1031.353,329.050,370.519,171.661,45.792,158.911
C03399=1031.361,329.298,370.483,171.667,45.793,158.911
C03400=1031.368,329.544,370.448,171.672,45.793,158.912
C03401=1031.375,329.792,370.412,171.676,45.794,158.913
C03402=1031.382,330.039,370.376,171.683,45.795,158.914
C03403=1031.389,330.287,370.341,171.687,45.796,158.915
C03404=1031.396,330.534,370.305,171.693,45.797,158.915
C03405=1031.404,330.782,370.269,171.698,45.798,158.916
C03406=1031.412,331.028,370.234,171.704,45.798,158.917
C03407=1031.419,331.277,370.199,171.709,45.800,158.918
C03408=1031.426,331.523,370.163,171.715,45.800,158.919
C03409=1031.433,331.771,370.127,171.720,45.801,158.919
C03410=1031.441,332.018,370.091,171.726,45.802,158.920
C03411=1031.448,332.266,370.055,171.731,45.803,158.921
C03412=1031.455,332.513,370.020,171.736,45.804,158.922
C03413=1031.463,332.760,369.984,171.742,45.805,158.923
C03414=1031.470,333.008,369.948,171.747,45.806,158.923
C03415=1031.477,333.255,369.912,171.753,45.807,158.924
C03416=1031.486,333.502,369.877,171.759,45.808,158.925
C03417=1031.493,333.749,369.841,171.764,45.809,158.926
C03418=1031.500,333.996,369.805,171.770,45.810,158.927
C03419=1031.508,334.245,369.769,171.775,45.810,158.928
C03420=1031.515,334.491,369.733,171.781,45.812,158.928
C03421=1031.522,334.739,369.697,171.786,45.813,158.929
C03422=1031.534,335.145,369.638,171.795,45.814,158.931
C03423=1031.546,335.551,369.578,171.804,45.816,158.932
C03424=1031.559,335.958,369.519,171.813,45.818,158.934
C03425=1031.571,336.364,369.459,171.822,45.820,158.935
C03426=1031.578,336.612,369.423,171.828,45.821,158.936
C03427=1031.585,336.858,369.387,171.833,45.822,158.937
C03428=1031.592,337.106,369.351,171.840,45.823,158.938
C03429=1031.600,337.354,369.314,171.844,45.824,158.938
C03430=1031.608,337.600,369.277,171.851,45.825,158.939
C03431=1031.615,337.847,369.242,171.856,45.827,158.940
C03432=1031.623,338.095,369.205,171.862,45.827,158.941
C03433=1031.630,338.342,369.169,171.867,45.829,158.942
C03434=1031.637,338.590,369.132,171.873,45.830,158.943
C03435=1031.645,338.837,369.096,171.879,45.831,158.944
C03436=1031.652,339.083,369.060,171.884,45.832,158.945
C03437=1031.660,339.331,369.023,171.890,45.833,158.946
C03438=1031.668,339.578,368.987,171.896,45.834,158.947
C03439=1031.676,339.825,368.950,171.901,45.836,158.948
C03440=1031.683,340.073,368.913,171.908,45.837,158.949
C03441=1031.690,340.320,368.877,171.912,45.838,158.949
C03442=1031.698,340.567,368.840,171.919,45.839,158.950
C03443=1031.706,340.815,368.804,171.925,45.840,158.951
C03444=1031.712,341.062,368.768,171.930,45.842,158.952
C03445=1031.720,341.308,368.731,171.936,45.843,158.953
C03446=1031.728,341.556,368.694,171.942,45.844,158.954
C03447=1031.735,341.803,368.657,171.947,45.846,158.955
C03448=1031.743,342.050,368.621,171.954,45.847,158.956
C03449=1031.750,342.298,368.583,171.960,45.848,158.957
C03450=1031.758,342.544,368.546,171.965,45.849,158.958
C03451=1031.765,342.792,368.509,171.971,45.851,158.959
C03452=1031.773,343.039,368.472,171.977,45.852,158.960
C03453=1031.781,343.286,368.436,171.982,45.853,158.961
C03454=1031.788,343.534,368.399,171.989,45.855,158.962
C03455=1031.796,343.780,368.362,171.995,45.856,158.963
C03456=1031.803,344.028,368.324,172.000,45.858,158.964
C03457=1031.811,344.275,368.288,172.006,45.859,158.965
C03458=1031.818,344.522,368.250,172.012,45.860,158.966
C03459=1031.826,344.769,368.214,172.019,45.861,158.967
C03460=1031.833,345.016,368.176,172.024,45.863,158.968
C03461=1031.841,345.263,368.139,172.030,45.864,158.969
C03462=1031.849,345.510,368.102,172.036,45.866,158.970
C03463=1031.856,345.757,368.065,172.042,45.867,158.971
C03464=1031.864,346.005,368.028,172.048,45.869,158.972
C03465=1031.872,346.252,367.991,172.054,45.870,158.973
C03466=1031.879,346.499,367.953,172.060,45.871,158.974
C03467=1031.887,346.746,367.916,172.067,45.873,158.975
C03468=1031.895,346.993,367.879,172.072,45.874,158.976
C03469=1031.903,347.240,367.842,172.078,45.876,158.977
C03470=1031.910,347.487,367.804,172.084,45.877,158.978
C03471=1031.918,347.735,367.767,172.091,45.879,158.979
C03472=1031.926,347.982,367.729,172.097,45.880,158.980
C03473=1031.934,348.229,367.692,172.102,45.882,158.981
C03474=1031.941,348.475,367.654,172.109,45.884,158.982
C03475=1031.948,348.722,367.617,172.115,45.885,158.983
C03476=1031.957,348.970,367.579,172.121,45.887,158.984
C03477=1031.964,349.217,367.542,172.127,45.888,158.985
C03478=1031.976,349.620,367.480,172.138,45.891,158.987
C03479=1031.990,350.023,367.419,172.147,45.893,158.989
C03480=1032.002,350.426,367.357,172.157,45.896,158.991
C03481=1032.015,350.829,367.296,172.167,45.898,158.992
C03482=1032.022,351.076,367.257,172.173,45.900,158.993
C03483=1032.030,351.323,367.220,172.180,45.902,158.994
C03484=1032.038,351.570,367.181,172.186,45.904,158.996
C03485=1032.046,351.817,367.144,172.192,45.905,158.997
C03486=1032.053,352.063,367.106,172.199,45.907,158.998
C03487=1032.061,352.311,367.068,172.205,45.908,158.999
C03488=1032.069,352.558,367.030,172.211,45.910,159.000
C03489=1032.077,352.806,366.992,172.217,45.912,159.001
C03490=1032.085,353.052,366.954,172.224,45.914,159.002
C03491=1032.092,353.299,366.917,172.230,45.915,159.003
C03492=1032.100,353.546,366.878,172.236,45.917,159.004
C03493=1032.108,353.793,366.840,172.243,45.919,159.006
C03494=1032.116,354.040,366.802,172.249,45.920,159.007
C03495=1032.124,354.287,366.765,172.256,45.922,159.008
C03496=1032.132,354.534,366.726,172.262,45.924,159.009
C03497=1032.140,354.780,366.688,172.269,45.926,159.010
C03498=1032.148,355.028,366.649,172.275,45.927,159.011
C03499=1032.155,355.275,366.612,172.281,45.929,159.013
C03500=1032.164,355.522,366.574,172.288,45.931,159.014
C03501=1032.171,355.768,366.535,172.294,45.933,159.015
C03502=1032.180,356.015,366.497,172.301,45.934,159.016
C03503=1032.188,356.263,366.458,172.307,45.936,159.017
C03504=1032.195,356.509,366.420,172.314,45.939,159.018
C03505=1032.203,356.756,366.381,172.320,45.940,159.020
C03506=1032.211,357.003,366.343,172.327,45.942,159.021
C03507=1032.219,357.250,366.304,172.333,45.944,159.022
C03508=1032.227,357.497,366.266,172.340,45.946,159.023
C03509=1032.235,357.744,366.227,172.346,45.948,159.024
C03510=1032.243,357.991,366.189,172.353,45.950,159.026
C03511=1032.250,358.237,366.149,172.359,45.951,159.027
C03512=1032.258,358.484,366.111,172.366,45.954,159.028
C03513=1032.266,358.732,366.072,172.373,45.956,159.029
C03514=1032.274,358.978,366.034,172.379,45.957,159.030
C03515=1032.282,359.225,365.995,172.386,45.960,159.032
C03516=1032.291,359.472,365.956,172.392,45.961,159.033
C03517=1032.299,359.719,365.917,172.400,45.964,159.034
C03518=1032.306,359.966,365.879,172.406,45.965,159.035
C03519=1032.315,360.212,365.840,172.413,45.967,159.037
C03520=1032.323,360.459,365.801,172.420,45.969,159.038
C03521=1032.331,360.706,365.762,172.426,45.971,159.039
C03522=1032.339,360.953,365.724,172.433,45.974,159.040
C03523=1032.347,361.200,365.685,172.440,45.976,159.042
C03524=1032.355,361.447,365.645,172.446,45.978,159.043
C03525=1032.363,361.693,365.606,172.454,45.980,159.044
C03526=1032.371,361.941,365.567,172.460,45.982,159.046
C03527=1032.378,362.187,365.528,172.467,45.984,159.047
C03528=1032.387,362.434,365.489,172.474,45.986,159.048
C03529=1032.395,362.681,365.450,172.480,45.988,159.049
C03530=1032.403,362.927,365.410,172.487,45.991,159.051
C03531=1032.411,363.174,365.370,172.495,45.992,159.052
C03532=1032.419,363.421,365.332,172.501,45.995,159.053
C03533=1032.427,363.667,365.292,172.508,45.997,159.055
C03534=1032.440,364.077,365.227,172.520,46.001,159.057
C03535=1032.454,364.486,365.162,172.531,46.004,159.059
C03536=1032.468,364.896,365.096,172.542,46.008,159.061
C03537=1032.481,365.304,365.030,172.554,46.011,159.063
C03538=1032.490,365.551,364.991,172.561,46.014,159.065
C03539=1032.498,365.798,364.951,172.568,46.016,159.066
C03540=1032.506,366.045,364.912,172.575,46.018,159.068
C03541=1032.514,366.291,364.872,172.582,46.020,159.069
C03542=1032.522,366.538,364.833,172.589,46.023,159.070
C03543=1032.531,366.785,364.793,172.596,46.025,159.072
C03544=1032.538,367.032,364.753,172.604,46.028,159.073
C03545=1032.547,367.278,364.714,172.611,46.030,159.074
C03546=1032.555,367.525,364.675,172.617,46.032,159.076
C03547=1032.564,367.772,364.634,172.625,46.035,159.077
C03548=1032.572,368.018,364.594,172.632,46.037,159.079
C03549=1032.581,368.265,364.555,172.639,46.039,159.080
C03550=1032.589,368.512,364.515,172.647,46.042,159.081
C03551=1032.597,368.758,364.475,172.653,46.044,159.083
C03552=1032.605,369.005,364.435,172.660,46.046,159.084
C03553=1032.614,369.252,364.396,172.668,46.049,159.086
C03554=1032.623,369.498,364.355,172.675,46.051,159.087
C03555=1032.631,369.745,364.316,172.683,46.053,159.088
C03556=1032.639,369.991,364.275,172.690,46.056,159.090
C03557=1032.648,370.238,364.235,172.696,46.059,159.091
C03558=1032.656,370.485,364.195,172.705,46.061,159.093
C03559=1032.663,370.732,364.155,172.711,46.064,159.094
C03560=1032.672,370.978,364.115,172.719,46.066,159.096
C03561=1032.680,371.224,364.074,172.726,46.069,159.097
C03562=1032.689,371.471,364.034,172.733,46.071,159.099
C03563=1032.697,371.717,363.994,172.741,46.074,159.100
C03564=1032.705,371.964,363.953,172.748,46.076,159.102
C03565=1032.714,372.211,363.912,172.756,46.079,159.103
C03566=1032.722,372.457,363.871,172.763,46.082,159.105
C03567=1032.730,372.704,363.832,172.771,46.085,159.106
C03568=1032.739,372.951,363.791,172.778,46.087,159.108
C03569=1032.747,373.197,363.750,172.786,46.089,159.109
C03570=1032.756,373.443,363.710,172.793,46.092,159.111
C03571=1032.765,373.690,363.669,172.801,46.095,159.112
C03572=1032.773,373.936,363.629,172.808,46.098,159.114
C03573=1032.782,374.183,363.588,172.816,46.100,159.115
C03574=1032.790,374.429,363.548,172.823,46.103,159.117
C03575=1032.799,374.676,363.507,172.831,46.105,159.118
C03576=1032.807,374.922,363.466,172.839,46.108,159.120
C03577=1032.816,375.169,363.426,172.846,46.111,159.122
C03578=1032.824,375.415,363.385,172.854,46.114,159.123
C03579=1032.833,375.662,363.344,172.861,46.116,159.125
C03580=1032.842,375.908,363.303,172.869,46.119,159.126
C03581=1032.850,376.155,363.262,172.877,46.122,159.128
C03582=1032.858,376.401,363.222,172.884,46.124,159.129
C03583=1032.867,376.648,363.181,172.893,46.128,159.131
C03584=1032.877,376.894,363.140,172.901,46.130,159.133
C03585=1032.885,377.140,363.099,172.908,46.133,159.134
C03586=1032.893,377.387,363.058,172.916,46.136,159.136
C03587=1032.902,377.634,363.016,172.924,46.138,159.137
C03588=1032.911,377.880,362.976,172.931,46.141,159.139
C03589=1032.920,378.126,362.934,172.939,46.144,159.141
C03590=1032.927,378.344,362.898,172.946,46.147,159.142
C03591=1032.935,378.562,362.862,172.953,46.150,159.144
C03592=1032.942,378.780,362.825,172.960,46.152,159.145
C03593=1032.950,378.997,362.788,172.967,46.155,159.146
C03594=1032.958,379.215,362.751,172.974,46.158,159.148
C03595=1032.965,379.433,362.715,172.981,46.160,159.149
C03596=1032.972,379.651,362.679,172.988,46.163,159.151
C03597=1032.980,379.869,362.642,172.995,46.165,159.152
C03598=1032.989,380.115,362.600,173.003,46.168,159.154
C03599=1032.998,380.362,362.558,173.011,46.171,159.156
C03600=1033.006,380.607,362.517,173.018,46.174,159.157
C03601=1033.015,380.854,362.475,173.027,46.177,159.159
C03602=1033.024,381.100,362.434,173.035,46.180,159.161
C03603=1033.033,381.347,362.393,173.043,46.184,159.163
C03604=1033.042,381.594,362.351,173.051,46.186,159.164
C03605=1033.051,381.840,362.309,173.059,46.190,159.166
C03606=1033.059,382.086,362.268,173.067,46.193,159.168
C03607=1033.068,382.332,362.226,173.075,46.196,159.170
C03608=1033.076,382.579,362.184,173.083,46.199,159.171
C03609=1033.085,382.824,362.141,173.092,46.202,159.173
C03610=1033.094,383.068,362.100,173.100,46.205,159.175
C03611=1033.103,383.312,362.058,173.108,46.208,159.176
C03612=1033.111,383.555,362.018,173.116,46.211,159.178
C03613=1033.120,383.798,361.976,173.124,46.215,159.180
C03614=1033.129,384.042,361.935,173.133,46.218,159.182
C03615=1033.138,384.286,361.893,173.141,46.220,159.183
C03616=1033.147,384.529,361.851,173.149,46.223,159.185
C03617=1033.156,384.773,361.810,173.157,46.227,159.187
C03618=1033.165,385.019,361.768,173.166,46.230,159.189
C03619=1033.174,385.265,361.726,173.174,46.234,159.191
C03620=1033.183,385.512,361.684,173.183,46.237,159.192
C03621=1033.193,385.757,361.642,173.191,46.240,159.194
C03622=1033.201,386.004,361.600,173.200,46.243,159.196
C03623=1033.211,386.249,361.558,173.208,46.247,159.198
C03624=1033.220,386.497,361.516,173.217,46.250,159.200
C03625=1033.229,386.742,361.473,173.225,46.253,159.201
C03626=1033.238,386.988,361.430,173.233,46.256,159.203
C03627=1033.247,387.235,361.388,173.242,46.260,159.205
C03628=1033.257,387.481,361.346,173.250,46.263,159.207
C03629=1033.266,387.727,361.303,173.259,46.267,159.209
C03630=1033.274,387.974,361.261,173.267,46.270,159.211
C03631=1033.283,388.219,361.218,173.276,46.273,159.213
C03632=1033.293,388.466,361.176,173.284,46.277,159.215
C03633=1033.302,388.712,361.133,173.293,46.280,159.216
C03634=1033.311,388.958,361.090,173.302,46.284,159.218
C03635=1033.320,389.204,361.047,173.311,46.287,159.220
C03636=1033.329,389.450,361.004,173.320,46.291,159.222
C03637=1033.339,389.696,360.962,173.329,46.294,159.224
